// TwinCAT 3 PLC project Lamp
// Title: ESO LDC Lamp Library
// Company: ESO
// Author: Dan Popovic
// ProjectVersion: 1.1.1.6
// Description: Local Device Control - LDC Lamp Library based on State Machine
// ProgramVersion: 3.1.0.8
// libraries:
//   Tc2_Standard, * (Beckhoff Automation GmbH)
//   Tc2_System, * (Beckhoff Automation GmbH)
//   Tc3_EventLogger, * (Beckhoff Automation GmbH)
//   Tc3_Module, * (Beckhoff Automation GmbH)
//   VisuDialogs, * (System)
//   VisuSymbols,3.5.10.0,System
// project tree:
//   DUTs/Enumerated/ E_LAMP_COMMAND.TcDUT, E_LAMP_RPC_ERROR.TcDUT, E_LAMP_EVENT.TcDUT, E_LAMP_ERROR.TcDUT, E_LAMP_STATUS.TcDUT, E_LAMP_STATE.TcDUT, E_LAMP_HW_STATUS.TcDUT, E_LAMP_SUBSTATE.TcDUT
//   DUTs/Structures/ T_LAMP_CFG.TcDUT, T_SIM_LAMP_CFG.TcDUT, T_LAMP_CTRL.TcDUT, T_LAMP_INFO.TcDUT, T_LAMP_STAT.TcDUT, T_SIM_LAMP_STAT.TcDUT
//   / GlobalTextList.TcGTLO, PlcTask.TcTTO (not stored), Visualization Manager.TcVMO (not stored)
//   POUs/ FB_SIM_LAMP.TcPOU, FB_LAMP_BASE.TcPOU, FB_LAMP.TcPOU, MAIN.TcPOU
//   Version/ Global_Version.TcGVL
//   VISUs/ GUI_Lamp001.TcVIS, GUI_Lamp002.TcVIS
//   VISUs/Templates/ GUI_TEMPLATE_LAMP.TcVIS
// real-time tasks:
//   TASK PlcTask: cycle T#10ms, priority 20, ADS port 350
// variable links:
//   Lamp/Lamp Instance <-> Lamp/Lamp Instance
//     PlcTask Inputs/MAIN.Lamp001.i_bFault <-> PlcTask Outputs/MAIN.SIM_Lamp001.q_bFault
//     PlcTask Inputs/MAIN.Lamp002.i_bFault <-> PlcTask Outputs/MAIN.SIM_Lamp002.q_bFault
//     PlcTask Inputs/MAIN.Lamp001.i_bOn <-> PlcTask Outputs/MAIN.SIM_Lamp001.q_bOn
//     PlcTask Inputs/MAIN.Lamp002.i_bOn <-> PlcTask Outputs/MAIN.SIM_Lamp002.q_bOn
//     PlcTask Inputs/MAIN.Lamp001.i_nCouplerState <-> PlcTask Outputs/MAIN.SIM_Lamp001.q_nCouplerState
//     PlcTask Inputs/MAIN.Lamp002.i_nCouplerState <-> PlcTask Outputs/MAIN.SIM_Lamp002.q_nCouplerState
//     PlcTask Inputs/MAIN.Lamp001.i_nOn <-> PlcTask Outputs/MAIN.SIM_Lamp001.q_nOn
//     PlcTask Inputs/MAIN.Lamp002.i_nOn <-> PlcTask Outputs/MAIN.SIM_Lamp002.q_nOn
//     PlcTask Inputs/MAIN.SIM_Lamp001.i_bSwitch <-> PlcTask Outputs/MAIN.Lamp001.q_bSwitch
//     PlcTask Inputs/MAIN.SIM_Lamp002.i_bSwitch <-> PlcTask Outputs/MAIN.Lamp002.q_bSwitch

// ---- DUTs/Enumerated/E_LAMP_COMMAND.TcDUT
{attribute 'qualified_only'}
{attribute 'strict'}
TYPE E_LAMP_COMMAND :
(
	NONE	:= 0,
	
	RESET,
	INIT,
	STOP,
	ENABLE,
	DISABLE,
	ON,
	OFF
	
);
END_TYPE

// ---- DUTs/Enumerated/E_LAMP_RPC_ERROR.TcDUT
{attribute 'qualified_only'}
{attribute 'strict'}
TYPE E_LAMP_RPC_ERROR :
(
	OK						:= 0,
	NOT_OP					:= -1,			
	NOT_NOTOP_READY			:= -2,			
	NOT_NOTOP_NOTREADY		:= -3,			
	SWITCHING_ON			:= -4,			
	SWITCHING_OFF			:= -5,			
	COOLING					:= -6,			
	LOCAL					:= -7			
);
END_TYPE

// ---- DUTs/Enumerated/E_LAMP_EVENT.TcDUT
{attribute 'qualified_only'}
{attribute 'strict'}
TYPE E_LAMP_EVENT :
(
	NONE	:= 0,
	
	(* events corresponding to commands *)
	RESET,
	INIT,
	STOP,
	ENABLE,
	DISABLE,
	ON,
	OFF,
	
	(* 
		Events corresponding to internal events 
	*)
	
	INITON,		// Needed for detection of HW failures during initialisation
	INITOFF,
	DISABLEON,
	DISABLEOFF,
	WARMED_UP,
	COOLED_DOWN,
	LIMIT_ON,	// Time ON limit has been exceeded
	
	(* events mapped to HW signals *)
	ISON,
	ISOFF,

	HWOK,
	ERRHW,
	ERRMAXON,
	ERRFAULT,
	ERRINIT,
	ERRDISABLE,
	ERRTIMEOUTOFF,
	ERRTIMEOUTON
	
);
END_TYPE

// ---- DUTs/Enumerated/E_LAMP_ERROR.TcDUT
{attribute 'qualified_only'}
{attribute 'strict'}
TYPE E_LAMP_ERROR :
(
	OK					:= 0,
	HW_NOT_OP,			
	INIT_FAILURE,		
	UNEXPECTED_OFF,
	UNEXPECTED_ON,
	FAULT_SIG,
	MAXON,
	STILL_COOLING,
	TIMEOUT_DISABLE,
	TIMEOUT_INIT,
	TIMEOUT_OFF,
	TIMEOUT_ON,
	// Simulator errors
	SIM_NOT_INITIALISED	:= 90,
	SIM_NULL_POINTER		:= 100	
);
END_TYPE

// ---- DUTs/Enumerated/E_LAMP_STATUS.TcDUT
{attribute 'qualified_only'}
{attribute 'strict'}
TYPE E_LAMP_STATUS :
(
	OK	:= 0,
	ERROR
);
END_TYPE

// ---- DUTs/Enumerated/E_LAMP_STATE.TcDUT
{attribute 'qualified_only'}
{attribute 'strict'}
TYPE E_LAMP_STATE :
(
	NONE	:= 0,
	NOTOP,
	OP
);
END_TYPE

// ---- DUTs/Enumerated/E_LAMP_HW_STATUS.TcDUT
{attribute 'qualified_only'}
{attribute 'strict'}
TYPE E_LAMP_HW_STATUS :
(
	UNKNOWN	:= 0,
	ERROR,
	OFF,
	ON
);
END_TYPE

// ---- DUTs/Enumerated/E_LAMP_SUBSTATE.TcDUT
{attribute 'qualified_only'}
{attribute 'strict'}
TYPE E_LAMP_SUBSTATE :
(
	NONE				:= 0,
	
	NOTOP_NOTREADY		:= 100,
	NOTOP_INITIALIZING	:= 102,
	NOTOP_READY_OFF		:= 103,
	NOTOP_READY_ON		:= 104,
	NOTOP_ERROR			:= 199,
	
	OP_DISABLING		:= 205,
	OP_OFF				:= 206,            
	OP_SWITCHING_OFF	:= 207,           
	OP_COOLING			:= 208,
	OP_ON				:= 209,
	OP_SWITCHING_ON		:= 210,
	OP_WARMING			:= 211,
	OP_ERROR			:= 299
);
END_TYPE

// ---- DUTs/Structures/T_LAMP_CFG.TcDUT
TYPE T_LAMP_CFG :
STRUCT
	sName:				STRING	:= 'Lamp';	// Instance name
	bActiveLowFault:	BOOL 	:= FALSE;	(* If TRUE, Fault signal is Active Low *)
	bActiveLowOn:		BOOL 	:= FALSE;	(* If TRUE, On signal is Active Low *)
	bActiveLowSwitch:	BOOL 	:= FALSE;	(* If TRUE, Switch ctrl signal is Active Low *)

	bIgnoreFault:		BOOL 	:= FALSE;	(* If TRUE, Fault feedback signal is ignored *)
	bInitialState:		BOOL 	:= FALSE;	(* default lamp state is OFF *)
	bInvertAnalog:		BOOL 	:= FALSE;	(* If TRUE, analog feedback is active, if signal < nAnalogThreshold *)
	
	lrInitialIntensity:	LREAL 	:= 0.0;		// Initial intensity [%]. Default 0.0.

	nAnalogThreshold:	DINT 	:= 0;		(* Analog feedback signal threshold [bits].
										  	If this signal is used, any value above it will indicate that the lamp is ON. *)
	nFullRange:			UDINT 	:= 32767;	(* Full range of A/D converter for analog output for intensity control. Default is 15-bit.
										  	Beckhoff 16-bit analog output terminals include the sign.
										  	Effectively, for 0-10V terminals, this is a 15-bit resolution.  *)
	nSigStablePeriod:   UDINT 	:= 100;		(* signal is stable if it has been constant for so long [msec] *)
	nTimeout:     		UDINT 	:= 3000;	(* timeout for transitions [msec] *)


	nCooldown:			UDINT 	:= 0;		(* Cooldown time [sec] *)
	nMaxOn:				UDINT 	:= 0;		(* Maximum time for lamp to be ON [sec]. Zero means no limit. *)
	nWarmup:			UDINT 	:= 0;		(* Warmup time [sec] *)
	
	// Logging
	bLogExtTime:		BOOL 	:= FALSE;		// If TRUE, use external time in event logs. Default FALSE.
	bDebug:				BOOL 	:= FALSE;		// If TRUE, show event logs of Debug type. Default FALSE.
	bLog:				BOOL 	:= TRUE;		// If TRUE, log events. Default TRUE.
	
END_STRUCT
END_TYPE

// ---- DUTs/Structures/T_SIM_LAMP_CFG.TcDUT
TYPE T_SIM_LAMP_CFG :
STRUCT
	bActiveLowFault:	BOOL := FALSE;
	bActiveLowOn:		BOOL := FALSE;
	bActiveLowSwitch:	BOOL := FALSE;

	bInvertAnalog:		BOOL := FALSE;	// If TRUE, analog feedback is active, if signal < nAnalogThreshold
	
	nAnalogThreshold:	DINT := 0;		// Analog feedback signal threshold [bits].
	nDelay:     		UDINT := 1000;	// Simulated delay for commands [msec]
	
END_STRUCT
END_TYPE

// ---- DUTs/Structures/T_LAMP_CTRL.TcDUT
TYPE T_LAMP_CTRL :
STRUCT
	nCommand:		E_LAMP_COMMAND	:= E_LAMP_COMMAND.NONE;	(* See E_LAMP_COMMAND *)
	lrIntensity: 	LREAL	:= 0.0;					(* Intensity 0-100% [%] *)
	nTimeOnLimit:	UDINT	:= 0;					(* Auto OFF after this time [sec]. 0 - no limit *)
	bExecute:		BOOL;
	
END_STRUCT
END_TYPE

// ---- DUTs/Structures/T_LAMP_INFO.TcDUT
TYPE T_LAMP_INFO :
STRUCT
(*
Driver Information 

Change Log:
	0.1	2016-07-07	- First version.
	0.2	2016-07-08	- Implemented warming up and cooling down.
					- Creation of Lamp.library.
					- Cleanup of code.
	0.3	2016-07-11	- Implemented time ON/OFF update.
					- Implemented MAXON protection.
	0.4	2016-07-11	- Addition of Configuration and Status in Template GUI.
					- Addition of Local Control in Template GUI.
	0.5	2016-07-11	- GUI buttons disabled if not in Local Mode.
	0.6	2016-07-12	- Corrected Time Update.
					- Corrected error handling and display.
	0.7 2017-01-30	- Addition of stat.sLastCommand.
					- Adopted Simulator from VLT FB_SIM_LAMP.
	0.8 2017-09-04	- Removed METHOD ActionDisableComplete.
					- Re-odered config and status parameters.
					- Improved checks returned values in RPC calls.
					- Addition of input parameter in_lrIntensity to RPC_On().
	0.9.0.0			- Single pointer to simulator
					- Updated Visualisation version
	0.10.0.0		- Simulator pointer renamed to ptrDev.
					- Additional checks in RPC_On/Off.
	0.11.0.0		- Corrected handling of intensity.
					- Addition of RPC Call Status in GUI template.
	0.12.0.0		- Corrected Simulator handling of Update.
					- Removed bUpdate variable from Simulator.
					- Errors cleared on ON and OFF commands.
	0.13.0.0		- Addition of all cfg params as input params.
					- Addition of M_Configure() in FB_LAMP_BASE.
					- Added return value for Simulator RPC calls.
					- Added small delay to simulator on re-boot.
					- Moved sName to cfg structure.
	0.14.0.0		- Addition of stat.sLibVersion
	0.15.0.0		- RPC calls return INT.
					- Addition of E_LAMP_RPC_ERROR.
	0.16.0.0		- Addition of M_GetErrorText().
					- M_SetStatus() replaced SetStatus().
					- Improved error handling.
	0.17.0.0		- Addition of M_GetRpcErrorText().
					- Addition of M_SetRpcStatus().
					- Improved template GUI.
	0.18.0.0		- Improved the State Machine to reflect HW State.
	0.18.0.1		- Tc2_System.F_GetSystemTime() used in GetTimeInSec().
					- Addition of library category ESO/ELT.
	0.19.0.0		- Renaming States STANDBY->NOTOP & FAILURE->ERROR.
					- RPC commands rejected in Local mode.
	0.20.0.0		- Addition of nTimeOnLimit control parameter.
	1.0.0.0			- WARNING: Requires TwinCAT 3.1 build 4022.20 or higher.
					- Projects need Tc3_EventLogger library included in References.
					- Addition of Methods for Event Logs.
					- Addition of method RPC_Debug().
	1.0.0.1			- Addition of cfg.bLog flag for enable/disable of logging.
					- Renamed RPC_Debug() to RPC_SetDebug().
					- Addition of RPC_SetLog().
	1.0.0.2			- Addition of {attribute 'OPC.UA.DA':='0'} before in_bLog declaration.
	1.0.0.3			- Compiled with TwinCAT 3.1 build 4022.27.
					- Renamed TC_EVENTS.OpsEventClass to TC_EVENTS.LampOpsEventClass.
					- Solved problem of 'growing' libraries by setting Property/Advanced/BuildAction to None for Lamp.library.
	1.1.0.0			- Using Strict enumerations.
*)
	sDate:			STRING(32)	:= '2019-04-24';
	sDescription:	STRING(80) 	:= 'State Machine based Lamp controller';
	sName:			STRING(64)	:= 'FB_LAMP';
	sPlatform:		STRING(32)	:= 'CoDeSys';
	sSynopsis:		STRING(64)	:= 'State Machine based Lamp controller';
	nVersionMajor:	DINT		:= 1;
	nVersionMinor:	DINT		:= 1;
END_STRUCT
END_TYPE

// ---- DUTs/Structures/T_LAMP_STAT.TcDUT
TYPE T_LAMP_STAT :
STRUCT
	//
	// Common variables START
	//
	bLocal:			BOOL	:= FALSE;						(* if TRUE, device operated from PLC GUI *)
	bCheckTimeLeft:	BOOL	:= FALSE;						(* if TRUE, check for max time is active *)
	bOnAnalog:		BOOL	:= FALSE;						(* if TRUE, analog  ON is active *)
	bOnDigital:		BOOL	:= FALSE;						(* if TRUE, digital ON is active *)

	nOn:			DINT		:= 0;		// Analog feedback [bit]
	
	nLastCommand:	E_LAMP_COMMAND	:= E_LAMP_COMMAND.NONE;		(* Last command sent to the device *)

	nErrorCode: 	E_LAMP_ERROR 	:= E_LAMP_ERROR.HW_NOT_OP;	(* Error code *)
	nHwStatus: 		E_LAMP_HW_STATUS:= E_LAMP_HW_STATUS.UNKNOWN;(* Unknown, error, on, of. See E_LAMP_HW_STATUS *)
	nRpcErrorCode: 	E_LAMP_RPC_ERROR:= E_LAMP_RPC_ERROR.OK;		(* RPC Error code *)
	nStatus: 		E_LAMP_STATUS	:= E_LAMP_STATUS.ERROR; 	(* Device status *)

	sErrorText: 	STRING 	:= 'OK'; 						(* Error text *)
	sHwStatus: 		STRING 	:= 'UNKNOWN'; 					(* HW Status in textual form: 'UNKNOWN', 'ERROR', 'OPEN' or 'CLOSED' *)
	sLastCommand:	STRING	:= 'NONE';						(* Last command, as string, sent to the device *)
	sLibVersion:	STRING	:= 'UNKNOWN';					(* Library version as string, e.g. '1.2.0.0' *)
	sRpcErrorText: 	STRING 	:= 'OK'; 						(* RPC Error text *)
	sStatus: 		STRING 	:= 'OK'; 						(* Status in textual form, e.g. 'OFF' *)
	
	sState:			STRING	:= 'NOT OP';
	sSubstate:		STRING	:= 'NOT READY';
	
	nState:			E_LAMP_STATE	:= E_LAMP_STATE.NOTOP;
	nSubstate:		E_LAMP_SUBSTATE	:= E_LAMP_SUBSTATE.NOTOP_NOTREADY;
	
	sActionDesc:	STRING	:= '';
	sEventDesc:		STRING	:= '';

	nCycleCounter:	UDINT	:= 0;							// Alive flag
	nCycleTime:		UDINT	:= 0;							// Cycle time in us (microsec)
	//
	// Common variables END
	//
	
	//
	// Device specific variables
	//
	lrIntensity: 		LREAL	:= 0.0; 	(* Intensity: 0-100% [%]*)

	nTimeLeft: 			UDINT 	:= 777;		(* Remaining Time before lamp is switched OFF [sec]. 777 means no limit. *)
	nTimeOn: 			UDINT 	:= 0;		(* Time lamp has been ON since last ON command [sec] *)
	nTimeOnLimit:		UDINT	:= 0;		(* Auto OFF after this time [sec]. 0 - no limit *)
	nTimeOnStart:		UDINT 	:= 0;		(* Absolute start time of last lamp ON command [sec] *)
	nTimeOnTotal:		UDINT 	:= 0;		(* Total time lamp has been ON [sec] *)
	nTimeOnTotalStart:	UDINT 	:= 0;		(* Absolute start time of lamp ON [sec] *)
	nTimeOff: 			UDINT 	:= 0;		(* Time lamp has been OFF [sec] *)
	nTimeOffStart:		UDINT 	:= 0;		(* Time lamp has been OFF [sec] *)
END_STRUCT
END_TYPE

// ---- DUTs/Structures/T_SIM_LAMP_STAT.TcDUT
TYPE T_SIM_LAMP_STAT :
STRUCT
	bInitialised:	BOOL	:= FALSE;						(* If TRUE, lamp simulator is initialised *)

	nErrorCode: 	E_LAMP_ERROR 	:= E_LAMP_ERROR.SIM_NOT_INITIALISED;	(* Error code *)
	sErrorText: 	STRING 	:= 'NOT INITIALISED'; 			(* Error text *)
	sStatus: 		STRING 	:= 'ERROR'; 					(* Lamp status in textual form, e.g. 'OFF' *)
END_STRUCT
END_TYPE

// ---- Version/Global_Version.TcGVL
{attribute 'TcGenerated'}
{attribute 'no-analysis'}
{attribute 'linkalways'}
// This function has been automatically generated from the project information.
VAR_GLOBAL CONSTANT
	{attribute 'const_non_replaced'}
	stLibVersion_ESO_LDC_Lamp_Library : ST_LibVersion := (iMajor := 1, iMinor := 1, iBuild := 1, iRevision := 6, nFlags := 0, sVersion := '1.1.1.6');
END_VAR

// ---- POUs/FB_SIM_LAMP.TcPOU
FUNCTION_BLOCK FB_SIM_LAMP
VAR_INPUT
	ptrDev:		POINTER TO FB_LAMP;
END_VAR
VAR_OUTPUT
END_VAR
VAR
	ptrCfg:		POINTER TO T_LAMP_CFG;
	ptrStat:	POINTER TO T_LAMP_STAT;

	{attribute 'OPC.UA.DA':='1'}
	cfg:			T_SIM_LAMP_CFG;		(* ActiveLow configuration for each signal *)
	{attribute 'OPC.UA.DA':='1'}
	stat:			T_SIM_LAMP_STAT;	(* Simulator status parameters *)
	
	{attribute 'OPC.UA.DA':='0'}
	bSwitch:		BOOL := FALSE;
	{attribute 'OPC.UA.DA':='0'}
	bSwitchLast:	BOOL := FALSE;
	
	{attribute 'OPC.UA.DA':='0'}
	bOn:			BOOL := TRUE;	// Digital feedback
	{attribute 'OPC.UA.DA':='0'}
	nOn:			DINT := 0;		// Analog feedback
	{attribute 'OPC.UA.DA':='0'}
	bFault:			BOOL := FALSE;
	{attribute 'OPC.UA.DA':='0'}
	nCouplerState:	UINT := 8;       // normal coupler state
	
    (* Inputs *)
	{attribute 'OPC.UA.DA':='0'}
	i_bSwitch 		AT %I*: 	BOOL;

	(* Outputs *)	
	{attribute 'OPC.UA.DA':='0'}
	q_bFault 		AT %Q*: 	BOOL;
	{attribute 'OPC.UA.DA':='0'}
	q_bOn 			AT %Q*: 	BOOL;	// Digital feedback signal
	{attribute 'OPC.UA.DA':='0'}
	q_nOn 			AT %Q*: 	INT;	// Analog feedback signal
	{attribute 'OPC.UA.DA':='0'}
	q_nCouplerState AT %Q*:		UINT := 8;
	
	{attribute 'OPC.UA.DA':='0'}
	timer:			TON;
	
	{attribute 'OPC.UA.DA':='0'}
	trigger:		R_TRIG;	// To capture device INIT

	{attribute 'OPC.UA.DA':='0'}
	counter:		DINT	:= 0; 	// Counter used to 	

	{attribute 'OPC.UA.DA':='0'}
	nOnStart:		DINT;
	{attribute 'OPC.UA.DA':='0'}
	nOnEnd:			DINT;
	{attribute 'OPC.UA.DA':='0'}
	nOnDelta:		DINT;		// Total analog signal change during ramp
	
	t1, t2:	LREAL;

END_VAR

// Give simulator 20 cycles of idle until real device is ready.
IF counter < 20 THEN
	counter	:= counter + 1;
	RETURN;
END_IF

// Initialise the simulator, i.e. set pointers to the real device, etc.
IF NOT stat.bInitialised THEN
	ptrCfg	:= ADR(ptrDev^.cfg);
	ptrStat	:= ADR(ptrDev^.stat);

	// Check for NULL pointers in input parameters
	IF ptrCfg = 0  OR  ptrStat = 0 THEN
		stat.nErrorCode	:= E_LAMP_ERROR.SIM_NULL_POINTER;
		stat.sErrorText	:= 'ERROR: Input parameter is a NULL pointer';
		stat.sStatus	:= 'ERROR';
		RETURN;
	END_IF

	RPC_ResetConfig();	// Copy configuration from device
	
	// Set analog feedback to a good starting level.
	M_SetAnalogFeedback();

	timer(IN:=FALSE);
	timer(IN:=TRUE,PT:=UDINT_TO_TIME(100));	// Update almost immediately

	stat.nErrorCode	:= E_LAMP_ERROR.OK;
	stat.sErrorText	:= 'OK';
	stat.sStatus	:= 'OK';
	
	stat.bInitialised	:= TRUE;
	RETURN;
END_IF

// There are two possible triggers: 
// 	- Detect device INIT (action = 'ActionInitExecute')
// 	- Activation of switch (change of i_bSwitch state)

// Check for INIT trigger
trigger(CLK:=(ptrStat^.sActionDesc = 'ActionInitExecute'));

// Get the state of control command
bSwitch := M_GetLogicalState(i_bSwitch, cfg.bActiveLowSwitch);

IF trigger.Q THEN
	timer(IN:=FALSE);
	RPC_ResetConfig();	// Copy configuration from device
	// Set analog feedback to a good starting level.
	M_SetAnalogFeedback();
ELSIF bSwitch <> bSwitchLast THEN
	ReloadConfig();	// Reload configuration from device
	
	// Switch value has changed. 
	bSwitchLast	:= bSwitch;

	// Delayed response
	timer(IN:=FALSE);
	timer(IN:=TRUE,PT:=UDINT_TO_TIME(cfg.nDelay));
	
	// If analog feedback is used, find out how much to ramp it.
	IF cfg.nAnalogThreshold <> 0	THEN
		nOnStart	:= nOn;
		// Set target feedback is 10 bit beyond the threshold.
		// This value depends on the command (on/off) and the logic (over/under threshold).
		IF bSwitch = M_GetLogicalState(TRUE, cfg.bActiveLowSwitch) THEN
		// The command was ON
			IF cfg.bInvertAnalog THEN
				nOnEnd	:= cfg.nAnalogThreshold - 10;
			ELSE
				nOnEnd	:= cfg.nAnalogThreshold + 10;
			END_IF
		ELSE
		// The command was OFF
			IF cfg.bInvertAnalog THEN
				nOnEnd	:= MAX(32000, cfg.nAnalogThreshold + 10);	// was cfg.nAnalogThreshold + 10;
			ELSE
				nOnEnd	:= 0;	// was cfg.nAnalogThreshold - 10;
			END_IF
		END_IF
		// This is how much to change simulated feedback over cfg.nDelay.
		nOnDelta	:= nOnEnd - nOnStart;
	END_IF
END_IF


// Execute the timer
timer();

// If analog feedback is used, ramp up/down the simulated feedback.
IF cfg.nAnalogThreshold <> 0	THEN
	bOn	:= FALSE;	// Don't use the digital feedback.
	IF timer.ET > INT_TO_TIME(0)	THEN
		t1	:= TIME_TO_LREAL(timer.ET);
		t2	:= TIME_TO_LREAL(timer.PT);
		nOn	:=	nOnStart + LREAL_TO_INT((t1*t1*t1) / (t2*t2*t2) * nOnDelta);
	END_IF
ELSE
	nOn	:= 0;
END_IF

// Set new outputs once the timer has expired
IF timer.Q THEN
	timer(IN:=FALSE);	// Reset timer
	// Set digital output, i.e. feedback, if analog feedback is not used.
	IF cfg.nAnalogThreshold = 0	THEN
		bOn	:= M_GetLogicalState(bSwitch,	cfg.bActiveLowOn);
	END_IF
END_IF


(* Assign outputs *)
q_bFault		:= M_GetLogicalState(bFault, cfg.bActiveLowFault);
q_bOn 			:= bOn;
q_nOn			:= DINT_TO_INT(nOn);
q_nCouplerState := nCouplerState;

METHOD M_GetLogicalState : BOOL
(*
	This method returns the state of the variable based on its 
	activeLow configuration.
	Syntax:
		bState	:= M_GetLogicalState (<var value>,  <activeLow cfg>);
		
	Example 1:
		var = TRUE;
		activeLow = FALSE;
		bState	:= M_GetLogicalState (TRUE,  FALSE); = TRUE

	Example 2:
		var = TRUE;
		activeLow = TRUE;
		bState	:= M_GetLogicalState (TRUE,  TRUE); = FALSE
*)
VAR_INPUT
	state:		BOOL;
	activeLow:	BOOL;
END_VAR
IF activeLow THEN
	M_GetLogicalState := NOT state;
ELSE
	M_GetLogicalState := state;
END_IF
END_METHOD

// Set starting analog feedback depending 
// on the analog feedback configuration and the command.
METHOD M_SetAnalogFeedback
VAR_INPUT
END_VAR
// Reset analog feedback, if not used.
IF cfg.nAnalogThreshold = 0	THEN
	nOn	:= 0;
ELSE
	// Analog feedback set to a value equivalent to OFF.
	IF cfg.bInvertAnalog THEN
		nOn	:= MAX(32000, cfg.nAnalogThreshold + 10);
	ELSE
		nOn	:= 0;
	END_IF
END_IF
END_METHOD

METHOD ReloadConfig : BOOL
VAR_INPUT
END_VAR
cfg.bActiveLowOn		:= ptrCfg^.bActiveLowOn;
cfg.bActiveLowFault		:= ptrCfg^.bActiveLowFault;
cfg.bActiveLowSwitch	:= ptrCfg^.bActiveLowSwitch;
cfg.bInvertAnalog		:= ptrCfg^.bInvertAnalog;
cfg.nDelay				:= ptrCfg^.nTimeout / 2;	// Response delay = 1/2 of real lamp timeout
cfg.nAnalogThreshold	:= ptrCfg^.nAnalogThreshold;
nCouplerState			:= 8;

// Reset analog feedback, if not used.
IF cfg.nAnalogThreshold = 0	THEN
	nOn	:= 0;
END_IF
END_METHOD

{attribute 'TcRpcEnable':='1'}
METHOD RPC_ResetConfig : INT
VAR_INPUT
END_VAR
ReloadConfig();

// Set valid intensity feedback
nOn	:= cfg.nAnalogThreshold;


// Reset Fault signal
bFault		:= FALSE;

// Get the Switch value
bSwitch := M_GetLogicalState(i_bSwitch, cfg.bActiveLowSwitch);

bOn	:= M_GetLogicalState(bSwitch,	cfg.bActiveLowOn);	// Set lamp state

RPC_ResetConfig	:= E_LAMP_RPC_ERROR.OK;
END_METHOD

{attribute 'TcRpcEnable':='1'}
METHOD RPC_SetActiveLow_Fault : INT
VAR_INPUT
	bValue:	BOOL;
END_VAR
cfg.bActiveLowFault	:= bValue;

RPC_SetActiveLow_Fault	:= E_LAMP_RPC_ERROR.OK;
END_METHOD

{attribute 'TcRpcEnable':='1'}
METHOD RPC_SetActiveLow_On : INT
VAR_INPUT
	bValue:	BOOL;
END_VAR
cfg.bActiveLowOn	:= bValue;

RPC_SetActiveLow_On	:= E_LAMP_RPC_ERROR.OK;
END_METHOD

{attribute 'TcRpcEnable':='1'}
METHOD RPC_SetActiveLow_Switch : INT
VAR_INPUT
	bValue:	BOOL;
END_VAR
cfg.bActiveLowSwitch	:= bValue;

RPC_SetActiveLow_Switch	:= E_LAMP_RPC_ERROR.OK;
END_METHOD

{attribute 'TcRpcEnable':='1'}
METHOD RPC_SetCouplerState : INT
VAR_INPUT
	nValue:	UINT;
END_VAR
nCouplerState	:= nValue;

RPC_SetCouplerState	:= E_LAMP_RPC_ERROR.OK;
END_METHOD

{attribute 'TcRpcEnable':='1'}
METHOD RPC_SetDelay : INT
VAR_INPUT
	nDelay:	UDINT;
END_VAR
cfg.nDelay	:= nDelay;

RPC_SetDelay	:= E_LAMP_RPC_ERROR.OK;
END_METHOD

{attribute 'TcRpcEnable':='1'}
METHOD RPC_SetFault : INT
VAR_INPUT
	bValue:	BOOL;
END_VAR
bFault	:= bValue;

RPC_SetFault	:= E_LAMP_RPC_ERROR.OK;
END_METHOD

END_FUNCTION_BLOCK

// ---- POUs/FB_LAMP.TcPOU
FUNCTION_BLOCK FB_LAMP EXTENDS FB_LAMP_BASE
VAR_INPUT
END_VAR
VAR_OUTPUT
END_VAR
VAR
	
	(***** Local variables *****)
	{attribute 'OPC.UA.DA' := '0'}
	bOn:		BOOL;	(* Feedback - combination of digital and analog *)
	{attribute 'OPC.UA.DA' := '0'}
	bFault: 	BOOL;
	{attribute 'OPC.UA.DA' := '0'}
	toutCmd:	TON;
	{attribute 'OPC.UA.DA' := '0'}
	trg:		R_TRIG;
	{attribute 'OPC.UA.DA' := '0'}
	timer:		TON;	(* Timer for measuring duration of events *)
	


	(***** Physical signals - to be mapped!!! *****)

	(* Outputs *)
	{attribute 'OPC.UA.DA' := '0'}
	q_bSwitch 		AT %Q*: 		BOOL;	(* Lamp control digital output *)
	{attribute 'OPC.UA.DA' := '0'}
	q_nIntensity 	AT %Q*: 		INT;	(* Analog OUT [bit] *)

	(* Inputs *)	
	{attribute 'OPC.UA.DA' := '0'}
	i_nCouplerState	AT %I*: 		UINT;	(* Link it to Coupler->InfoData->State *)
	{attribute 'OPC.UA.DA' := '0'}
	i_bFault 		AT %I*: 		BOOL;	(* HW fault signal *)
	{attribute 'OPC.UA.DA' := '0'}
	i_bOn 			AT %I*: 		BOOL;	(* Digital feedback signal *)
	{attribute 'OPC.UA.DA' := '0'}
	i_nOn			AT %I*: 		INT;	(* Analog feedback signal *)

END_VAR

// Execute the base class object FB_LAMP_BASE
SUPER^();

METHOD ActionDisableExecute
VAR_INPUT
END_VAR
SetAction('ActionDisableExecute');

// Log event
M_LogEventStart('DISABLE');

(* Set Lamp initial state obtained from the configuration *)
q_bSwitch			:= M_GetLogicalState(cfg.bInitialState, cfg.bActiveLowSwitch);
stat.lrIntensity	:= cfg.lrInitialIntensity;
q_nIntensity		:= LREAL_TO_INT(stat.lrIntensity / 100.0 * cfg.nFullRange);

(* start the cmd timer *)
toutCmd(IN:=FALSE);
toutCmd(IN:=TRUE,PT:=UDINT_TO_TIME(cfg.nTimeout));
END_METHOD

METHOD ActionEnableComplete
VAR_INPUT
END_VAR
SetAction('ActionEnableComplete');

// Log event
M_LogEventEnd('ENABLE');

(* reply OK *)
M_SetStatus(E_LAMP_ERROR.OK);

(* Reset the timer action *)
toutCmd(IN:=FALSE);
END_METHOD

METHOD ActionErrExecute
VAR
END_VAR
SetAction('ActionErrExecute');

IF nEvent = E_LAMP_EVENT.ERRFAULT THEN
	M_SetStatus(E_LAMP_ERROR.FAULT_SIG);
END_IF
END_METHOD

METHOD ActionInitAbort
VAR_INPUT
END_VAR
SetAction('ActionInitAbort');

M_SetStatus(E_LAMP_ERROR.OK);

(* Reset the timer for the command *)
toutCmd(IN:=FALSE);
END_METHOD

METHOD ActionInitComplete
VAR_INPUT
END_VAR
SetAction('ActionInitComplete');

// Log event
M_LogEventEnd('INIT');

(* reply OK *)
M_SetStatus(E_LAMP_ERROR.OK);

(* Reset the timer action *)
toutCmd(IN:=FALSE);
END_METHOD

METHOD ActionInitExecute
VAR_INPUT
END_VAR
VAR
	nCurrentTime:	UDINT;
END_VAR
SetAction('ActionInitExecute');

// Log event
M_LogEventStart('INIT');

M_SetStatus(E_LAMP_ERROR.OK);	// Clear any error

nCurrentTime			:= M_GetTimeInSec();
stat.nTimeOffStart		:= nCurrentTime;
M_UpdateTimes(bOnState:=FALSE, bRestart:=FALSE, bReset:=FALSE);


(* Set Lamp initial state obtained from the configuration *)
q_bSwitch			:= M_GetLogicalState(cfg.bInitialState, cfg.bActiveLowSwitch);
IF NOT cfg.bInitialState	THEN
	cfg.lrInitialIntensity	:= 0.0;
END_IF
stat.lrIntensity	:= cfg.lrInitialIntensity;
q_nIntensity		:= LREAL_TO_INT(stat.lrIntensity / 100.0 * cfg.nFullRange);

(* start the cmd timer *)
toutCmd(IN:=FALSE);
toutCmd(IN:=TRUE,PT:=UDINT_TO_TIME(cfg.nTimeout));
END_METHOD

METHOD ActionInitReject
VAR_INPUT
END_VAR
SetAction('ActionInitReject');

(* Reject an INIT command since another one is in progress. *)
(* do not reset the timer ... *)
END_METHOD

METHOD ActionMaxOnFailure
VAR_INPUT
END_VAR
(* code to initiate the switching OFF of the lamp *)
SetAction('ActionMaxOnFailure');

// Log event
M_LogEventError('Max ON time exceeded. Lamp switched OFF.');

(* Set the error *)
M_SetStatus(E_LAMP_ERROR.MAXON);

M_UpdateTimes(bOnState:=FALSE, bRestart:=TRUE, bReset:=FALSE);


(* Switch lamp OFF *)
q_bSwitch			:= M_GetLogicalState(FALSE, cfg.bActiveLowSwitch);
stat.lrIntensity	:= 0;
q_nIntensity		:= 0;


(* 
	Reset signal trigger and its timer. 
	Next transition activity, e.g. ActivitySwitchingOff, will complete when the signal has been OFF 
	for longer than cfg.nSigStablePeriod [ms].
*)
trg(CLK:=FALSE);
timer(IN:=FALSE);	// Timer for stable signal lasting cfg.nSigStablePeriod

(* Restart the command timer *)
toutCmd(IN:=FALSE);
toutCmd(IN:=TRUE,PT:=UDINT_TO_TIME(cfg.nTimeout));
END_METHOD

METHOD ActionOffExecute
VAR_INPUT
END_VAR
(* code to initiate the switching OFF of the lamp *)
SetAction('ActionOffExecute');

// Log event
M_LogEventStart('OFF');

(* Clear the error *)
M_SetStatus(E_LAMP_ERROR.OK);

M_UpdateTimes(bOnState:=FALSE, bRestart:=TRUE, bReset:=FALSE);


(* Switch lamp OFF *)
q_bSwitch			:= M_GetLogicalState(FALSE, cfg.bActiveLowSwitch);
stat.lrIntensity	:= 0;
q_nIntensity		:= 0;

(* 
	Reset signal trigger and its timer. 
	Next transition activity, e.g. ActivitySwitchingOff, will complete when the signal has been OFF 
	for longer than cfg.nSigStablePeriod [ms].
*)
trg(CLK:=FALSE);
timer(IN:=FALSE);	// Timer for stable signal lasting cfg.nSigStablePeriod

(* Restart the command timer *)
toutCmd(IN:=FALSE);
toutCmd(IN:=TRUE,PT:=UDINT_TO_TIME(cfg.nTimeout));
END_METHOD

METHOD ActionOnExecute
VAR_INPUT
END_VAR
(* Code to initiate turning the lamp ON *)

SetAction('ActionOnExecute');

// Log event
M_LogEventStart('ON');

(* Clear the error *)
M_SetStatus(E_LAMP_ERROR.OK);

(* Turn the control signal ON  and set the intensity *)
q_bSwitch			:= M_GetLogicalState(TRUE, cfg.bActiveLowSwitch);
stat.lrIntensity	:= ctrl.lrIntensity;
q_nIntensity		:= LREAL_TO_INT(stat.lrIntensity / 100.0 * cfg.nFullRange);

// Save time limit for ON and clear it from the command parameters
stat.nTimeOnLimit	:= ctrl.nTimeOnLimit;
ctrl.nTimeOnLimit	:= 0;


(* 
	Reset signal trigger and its timer. 
	Next transition activity, e.g. ActivitySwitchingOn, will complete when the signal has been ON 
	for longer than cfg.nSigStablePeriod [ms].
*)
trg(CLK:=FALSE);
timer(IN:=FALSE);	// Timer for stable signal lasting cfg.nSigStablePeriod

(* Start the timer for command timeout of cfg.nTimeout *)
toutCmd(IN:=FALSE);	
toutCmd(IN:=TRUE,PT:=UDINT_TO_TIME(cfg.nTimeout));
END_METHOD

METHOD ActionResetExecute
VAR_INPUT
END_VAR
SetAction('ActionResetExecute');

// Log event
M_LogEventEnd('RESET');

(* reply Error *)
M_SetStatus(E_LAMP_ERROR.OK);

(* Disable outputs *)
q_bSwitch			:= FALSE;
stat.lrIntensity	:= 0;
q_nIntensity		:= 0;

// Reset ON/OFF times
M_UpdateTimes(bOnState:=bOn,bRestart:=FALSE,bReset:=TRUE);	

(* Reset the timer for the command *)
toutCmd(IN:=FALSE);
END_METHOD

METHOD ActionUnexpExecute
VAR
END_VAR
SetAction('ActionUnexpExecute');

IF nEvent = E_LAMP_EVENT.ISON THEN
	// In case of a timeout while switching to ON the state after the timeout
	// will be E_LAMP_SUBSTATE.OP_OFF and later on the lamp will go ON. 
	// In this case, we don't want to set
	// the error to E_LAMP_ERROR.UNEXPECTED_ON but rather scilently
	// change the state to E_LAMP_SUBSTATE.OP_ON.
	IF 	stat.nErrorCode <> E_LAMP_ERROR.TIMEOUT_ON  AND
		stat.nErrorCode <> E_LAMP_ERROR.TIMEOUT_OFF 	THEN
		M_LogEventGeneral('Lamp unexpectedly switched ON');
		M_SetStatus(E_LAMP_ERROR.UNEXPECTED_ON);
	END_IF
ELSIF nEvent = E_LAMP_EVENT.ISOFF THEN
	// In case of a timeout while switching to OFF the state after the timeout
	// will be E_LAMP_SUBSTATE.OP_ON and later on the lamp will go OFF. 
	// In this case, we don't want to set
	// the error to E_LAMP_ERROR.UNEXPECTED_OFF but rather scilently
	// change the state to E_LAMP_SUBSTATE.OP_OFF.
	IF 	stat.nErrorCode <> E_LAMP_ERROR.TIMEOUT_OFF	AND
		stat.nErrorCode <> E_LAMP_ERROR.TIMEOUT_ON THEN
		M_LogEventGeneral('Lamp unexpectedly switched OFF');
		M_SetStatus(E_LAMP_ERROR.UNEXPECTED_OFF);
	END_IF
ELSIF nEvent = E_LAMP_EVENT.ON THEN
	// Clear time limit from the command parameters
	ctrl.nTimeOnLimit	:= 0;
	M_SetStatus(E_LAMP_ERROR.STILL_COOLING);
END_IF
END_METHOD

METHOD ActivityCoolingDown
VAR_INPUT
END_VAR
(* 
	This activity waits for cfg.nCooldown seconds until the lamp has warmed up.
	It triggers E_LAMP_EVENT.WARMED_UP event. 
*)
SetAction('ActivityCoolingDown');

// Update the OFF time
M_UpdateTimes(bOnState:=FALSE, bRestart:=FALSE, bReset:=FALSE);

(* 
	Warming is complete on expiration of the timer.
	If there is no warmup (cfg.nWarmup = 0), just set the event E_LAMP_EVENT.WARMED_UP.
*)
toutCmd();
IF 	toutCmd.Q OR 
	cfg.nCooldown = 0 OR
	(cfg.nCooldown > 0 AND stat.nTimeOff > cfg.nCooldown)	THEN
	// Log event
	M_LogEventEnd('OFF');

	toutCmd(IN:=FALSE);	(* Reset Timer *)
	
	nInternalEvent 		:= E_LAMP_EVENT.COOLED_DOWN;	// This will bring us to (E_LAMP_STATE.OP, E_LAMP_SUBSTATE.OP_OFF)
END_IF
END_METHOD

METHOD ActivityDisabling
VAR_INPUT
END_VAR
(* 
	Activity to monitor the lamp disabling task. 
	The end state should be the predefined position of the lamp
	that is defined by configuration parameter cfg.bInitialState.
*)
SetAction('ActivityDisabling');

(* check if the initial position is reached *)
IF cfg.bInitialState = FALSE THEN
	(* Waiting for OFF state *)
	IF	bOn   = FALSE THEN
		// Log event
		M_LogEventEnd('DISABLE_OFF');

		nEvent  := E_LAMP_EVENT.DISABLEOFF;
		M_SetStatus(E_LAMP_ERROR.OK);
		RETURN;
	END_IF
ELSE
	(* Waiting for ON state *)
	IF	bOn   = TRUE  THEN
		// Log event
		M_LogEventEnd('DISABLE_ON');

		nEvent  := E_LAMP_EVENT.DISABLEON;
		M_SetStatus(E_LAMP_ERROR.OK);
		RETURN;
	END_IF		
END_IF


(* 
	if the timeout is detected before reaching the target position, 
	then trigger the internal error event 
*)
toutCmd(IN:=TRUE);
IF toutCmd.Q THEN
	// Log event
	M_LogEventError('DISABLE command timed out');

	toutCmd(IN:=FALSE);	(* Reset the timer *)
	nInternalEvent  := E_LAMP_EVENT.ERRDISABLE;
	SetEvent(E_LAMP_ERROR.TIMEOUT_DISABLE);
END_IF
END_METHOD

METHOD ActivityInitializing
VAR_INPUT
END_VAR
(* 
	Activity to monitor the Lamp initialization task and 
	trigger the E_LAMP_EVENT.INITOFF or E_LAMP_EVENT.INITON event depending 
	on the configured default state. 		
*)
SetAction('ActivityInitializing');


(* 
	Check if the initial position is reached.
	We need additional internal events E_LAMP_EVENT.INITOFF & E_LAMP_EVENT.INITON in order to
	cope with the scenario when the initial state is the oposit one from the configured target.
	Example:
		The Lamp ISOFF at the beginning of this activity while the configured default state ISOFF.
		By introducing E_LAMP_EVENT.INITOFF & E_LAMP_EVENT.INITON we avoid the ISOFF event.
*)
IF cfg.bInitialState = FALSE THEN
	(* Waiting for OFF state *)
	IF	bOn   = FALSE THEN
		nInternalEvent  := E_LAMP_EVENT.INITOFF;
	END_IF
ELSE
	(* Waiting for ON state *)
	IF	bOn   = TRUE  THEN
		nInternalEvent  := E_LAMP_EVENT.INITON;
	END_IF		
END_IF


(* 
	If the timeout is detected before reaching the initial position, 
	then trigger the internal error event 
*)
toutCmd(IN:=TRUE);
IF toutCmd.Q THEN
	// Log event
	M_LogEventError('INIT command timed out');

	toutCmd(IN:=FALSE);	(* Reset the timer *)
	nInternalEvent  := E_LAMP_EVENT.ERRINIT;
	SetEvent(E_LAMP_ERROR.TIMEOUT_INIT);
END_IF
END_METHOD

METHOD ActivityOff
VAR_INPUT
END_VAR
SetAction('ActivityOff');

// Clear time limit for ON from the status
stat.nTimeOnLimit	:= 0;

// Update the OFF time
M_UpdateTimes(bOnState:=FALSE, bRestart:=FALSE, bReset:=FALSE);
END_METHOD

METHOD ActivityOn
VAR_INPUT
END_VAR
SetAction('ActivityOn');

// Update the ON time
M_UpdateTimes(bOnState:=TRUE, bRestart:=FALSE, bReset:=FALSE);

// Check if the lamp has been ON longer than the time limit for that command.
IF stat.nTimeOnLimit > 0 AND stat.nTimeOn > stat.nTimeOnLimit THEN
	M_LogEventGeneral('Time ON limit reached. Switching lamp OFF.');
	nEvent  := E_LAMP_EVENT.LIMIT_ON;
	RETURN;
END_IF
END_METHOD

METHOD ActivitySwitchingOff
VAR_INPUT
END_VAR
(* 
	This activity monitors the OFF lamp task and 
	triggers the ISOFF event at completion. 
*)
SetAction('ActivitySwitchingOff');


(* 
	The signal has to be OFF for longer than cfg.nSigStablePeriod [msec].
	The timer will start when bOn=FALSE trigger is detected.
*)
(* Execute trigger - note the 'NOT bOn' detectiong the transition from ON to OFF *)
trg(CLK := NOT bOn);

IF trg.Q THEN
	(* Restart the signal duration timer *)
	timer(IN:=FALSE);
	timer(IN:=TRUE,PT:=UDINT_TO_TIME(cfg.nSigStablePeriod));
END_IF

(* Execute signal duration timer *)
timer();

IF	timer.Q OR 
	((NOT bOn) AND cfg.nSigStablePeriod = 0) THEN
	timer(IN:=FALSE);	// Reset the signal duration timer
	toutCmd(IN:=FALSE);	// Reset the command timeout timer

	(* Update time ON/OFF *)
	M_UpdateTimes(bOnState:=TRUE, bRestart:=FALSE, bReset:=FALSE);

	(* 
		Normally, we would go to state E_LAMP_SUBSTATE.OP_COOLING. 
		However, if the cooldown time is zero, i.e. no cooldown, we go directly to state E_LAMP_SUBSTATE.OP_OFF.
	*)
	IF cfg.nCooldown > 0 THEN
		// Log event
		M_LogEventStart('COOLING');

		// Restart the command timeout timer
		toutCmd(IN:=TRUE,PT:=UDINT_TO_TIME(cfg.nCooldown * 1000));	// [sec] => [msec]
		nInternalEvent 		:= E_LAMP_EVENT.ISOFF;	// This will bring us to SetState(E_LAMP_STATE.OP, E_LAMP_SUBSTATE.OP_COOLING)
	ELSE
		// Log event
		M_LogEventEnd('OFF');

		nInternalEvent 		:= E_LAMP_EVENT.COOLED_DOWN;	// This will bring us to SetState(E_LAMP_STATE.OP, E_LAMP_SUBSTATE.OP_OFF)
	END_IF
	
//	M_SetStatus(E_LAMP_ERROR.OK);	

	RETURN;
END_IF

(* 
	if the timeout is detected before reaching the position, 
	then trigger the internal error event 
*)
toutCmd();
IF toutCmd.Q THEN
	toutCmd(IN:=FALSE);	(* Reset Timer *)
	timer(IN:=FALSE);	(* Reset the signal duration timer *)
	
	nInternalEvent  := E_LAMP_EVENT.ERRTIMEOUTOFF;
	SetEvent(E_LAMP_EVENT.ERRTIMEOUTOFF);
	M_SetStatus(E_LAMP_ERROR.TIMEOUT_OFF);	
END_IF
END_METHOD

METHOD ActivitySwitchingOn
VAR_INPUT
END_VAR
(* 
	This activity to monitor the ON lamp task and 
	trigger the ISON event at completion. 
*)
SetAction('ActivitySwitchingOn');

(* 
	The signal has to be ON for longer than cfg.nSigStablePeriod [msec].
	The timer will start when bOn trigger is detected.
*)
(* Execute trigger *)
trg(CLK:=bOn);

IF trg.Q THEN
	(* Restart the signal duration timer *)
	timer(IN:=FALSE);
	timer(IN:=TRUE,PT:=UDINT_TO_TIME(cfg.nSigStablePeriod));
END_IF

(* Execute signal duration timer *)
timer();

IF	timer.Q OR 
	(bOn AND cfg.nSigStablePeriod = 0) THEN
	timer(IN:=FALSE);	// Reset the signal duration timer
	toutCmd(IN:=FALSE);	// Reset the command timeout timer

	(* Update time ON/OFF *)
	IF stat.nTimeOn > 0 THEN
		// Lamp was already ON, restart the ON time.
		M_UpdateTimes(bOnState:=TRUE, bRestart:=TRUE, bReset:=FALSE);
	ELSE
		// Lamp was OFF, don't restart the ON time.
		M_UpdateTimes(bOnState:=TRUE, bRestart:=FALSE, bReset:=FALSE);
	END_IF

	(* 
		Normally, we would go to state E_LAMP_SUBSTATE.OP_WARMING. 
		However, if the warmup time is zero, i.e. no warmup, we go directly to state E_LAMP_SUBSTATE.OP_ON.
	*)
	IF cfg.nWarmup > 0 THEN
		// Log event
		M_LogEventStart('WARMING UP');

		// Restart the command timeout timer
		toutCmd(IN:=TRUE,PT:=UDINT_TO_TIME(cfg.nWarmup * 1000));	// [sec] => [msec]
		nInternalEvent 		:= E_LAMP_EVENT.ISON;	// This will bring us to SetState(E_LAMP_STATE.OP, E_LAMP_SUBSTATE.OP_WARMING)
	ELSE
		// Log event
		M_LogEventEnd('ON');

		nInternalEvent 		:= E_LAMP_EVENT.WARMED_UP;	// This will bring us to SetState(E_LAMP_STATE.OP, E_LAMP_SUBSTATE.OP_ON)
	END_IF
	
	M_SetStatus(E_LAMP_ERROR.OK);	

	RETURN;
END_IF

(* 
	if the timeout is detected before reaching the position, 
	then trigger the internal error event 
*)
toutCmd();
IF toutCmd.Q THEN
	// Log event
	M_LogEventError('ON command timed out');

	toutCmd(IN:=FALSE);	(* Reset Timer *)
	timer(IN:=FALSE);	(* Reset the signal duration timer *)
	
	nInternalEvent  := E_LAMP_EVENT.ERRTIMEOUTON;
	SetEvent(E_LAMP_EVENT.ERRTIMEOUTON);
	M_SetStatus(E_LAMP_ERROR.TIMEOUT_ON);	
END_IF
END_METHOD

METHOD ActivityWarmingUp
VAR_INPUT
END_VAR
(* 
	This activity waits for cfg.nWarmup seconds until the lamp has warmed up.
	It triggers E_LAMP_EVENT.WARMED_UP event. 
*)
SetAction('ActivityWarmingUp');

// Update the ON time
M_UpdateTimes(bOnState:=TRUE, bRestart:=FALSE, bReset:=FALSE);

(* 
	Warming is complete on expiration of the timer.
	If there is no warmup (cfg.nWarmup = 0), just set the event E_LAMP_EVENT.WARMED_UP.
*)
toutCmd();
IF toutCmd.Q OR cfg.nWarmup = 0 THEN
	// Log event
	M_LogEventEnd('ON');

	toutCmd(IN:=FALSE);	(* Reset Timer *)
	
	nInternalEvent 		:= E_LAMP_EVENT.WARMED_UP;	// This will bring us to (E_LAMP_STATE.OP, E_LAMP_SUBSTATE.OP_ON)
END_IF

// Check if the lamp has been ON longer than the time limit for that command.
IF stat.nTimeOnLimit > 0 AND stat.nTimeOn > stat.nTimeOnLimit THEN
	M_LogEventGeneral('Time ON limit reached during warmup. Switching lamp OFF.');
	nEvent  := E_LAMP_EVENT.LIMIT_ON;
	RETURN;
END_IF
END_METHOD

METHOD CheckForEvents
VAR_INPUT
END_VAR

(* 
	Start assuming the HW is OK. 
	This is needed to recover from the situation where 
	the HW was failing and now it is working.
*)
nEvent := E_LAMP_EVENT.HWOK;


(*
	Read all inputs, i.e. get status of INPUT signals based on ActiveLow configuration 
*)

bFault	:= M_GetLogicalState(i_bFault, cfg.bActiveLowFault) AND NOT cfg.bIgnoreFault;

(* The lamp ON feedback can be analog and/or digital. *)
stat.bOnDigital	:= M_GetLogicalState(i_bOn, cfg.bActiveLowOn);	// Digital feedback
stat.nOn		:= i_nOn;										// Analog  feedback

IF cfg.nAnalogThreshold <> 0	THEN
// Analog feedback is checked only if the threshold is not 0.0.
	stat.bOnAnalog	:=	((i_nOn > cfg.nAnalogThreshold) AND NOT cfg.bInvertAnalog) OR
						((i_nOn < cfg.nAnalogThreshold) AND     cfg.bInvertAnalog);
ELSE
	stat.bOnAnalog	:= FALSE;
END_IF
	
IF 	(stat.bOnDigital OR  stat.bOnAnalog)	THEN
	bOn	:= TRUE;
ELSE
	bOn	:= FALSE;
END_IF


M_UpdateTimes(bOnState:=bOn,bRestart:=FALSE, bReset:=FALSE);	// Update the Time


(* HW Status in textual form: 'ERROR', 'ON' or 'OFF' *)
IF 		bFault THEN
	stat.nHwStatus	:= E_LAMP_HW_STATUS.ERROR;
	stat.sHwStatus	:= 'ERROR';
ELSIF 	bOn   = TRUE  THEN
	stat.nHwStatus	:= E_LAMP_HW_STATUS.ON;
	stat.sHwStatus	:= 'ON';
ELSIF 	bOn   = FALSE  THEN
	stat.nHwStatus	:= E_LAMP_HW_STATUS.OFF;
	stat.sHwStatus	:= 'OFF';
END_IF

(* 
	Check for events in the following order: 
   	1) HW failure: without HW avilability there is no point to do anything
	2) Internal events: to allow completing the initiated commands before 
                        starting processing new commands. 
   	3) Commands: to react to external commands. Commands should be executed 
                 before processing HW signals to allow to start a recovery action.
   	4) HW signals:  such as Lamp is ON/OFF.
*)

IF 	i_nCouplerState <> 8 AND 
	NOT (ctrl.bExecute AND ctrl.nCommand = E_LAMP_COMMAND.RESET) THEN	
	// NOTE:	We give priority to RESET command in order 
	//			to be able to switch from OP to NOT_OP on RESET.
	(* Check if the HW is NOT OK *)
	(*
	If the hardware status is NOT OK, we cannot trust the readings.
	Variable i_nCouplerState has to be mapped to a State of a terminal, e.g. EK1100.
	The value should be 8.
 	*)
	SetEvent(E_LAMP_EVENT.ERRHW);
	M_SetStatus(E_LAMP_ERROR.HW_NOT_OP);

ELSIF nInternalEvent <> E_LAMP_EVENT.NONE THEN
	(* Handle internal events *)
	SetEvent(nInternalEvent);
	nInternalEvent := E_LAMP_EVENT.NONE;
ELSIF ctrl.bExecute = TRUE  THEN
	(* Handle commands *)
	ctrl.bExecute	:= FALSE;				(* Clear the Execute bit *)
	M_SetLastCommand(ctrl.nCommand);		(* Save the last command *)
	SetEvent(ctrl.nCommand);				(* Set the event *)
	ctrl.nCommand 	:= E_LAMP_COMMAND.NONE;	(* Clear the Command *)
ELSE
	(* Handle HW problems and unexpected bahaviour *)
	
	IF bFault THEN
		SetEvent(E_LAMP_EVENT.ERRFAULT);
		M_SetStatus(E_LAMP_ERROR.FAULT_SIG);
		RETURN;	
	END_IF

	IF stat.nSubstate = E_LAMP_SUBSTATE.NOTOP_READY_OFF OR 
	   stat.nSubstate = E_LAMP_SUBSTATE.NOTOP_READY_ON OR 
	   stat.nSubstate = E_LAMP_SUBSTATE.OP_DISABLING OR 
	   stat.nSubstate = E_LAMP_SUBSTATE.OP_OFF OR 
	   stat.nSubstate = E_LAMP_SUBSTATE.OP_ON	OR 
	   stat.nSubstate = E_LAMP_SUBSTATE.OP_ERROR THEN
	   
		(* Set events for ON and OFF *)		
		IF	bOn   = TRUE  THEN
			SetEvent(E_LAMP_EVENT.ISON);
		ELSIF	bOn   = FALSE THEN
			SetEvent(E_LAMP_EVENT.ISOFF);
		END_IF	
	END_IF	
(*
	IF stat.nSubstate = E_LAMP_SUBSTATE.OP_SWITCHING_ON THEN
		(* Set events for ON  *)		
		IF	bOn   = TRUE  THEN
			SetEvent(E_LAMP_EVENT.ISON);
		END_IF	
	END_IF	
	*)
END_IF
END_METHOD

METHOD M_GetRpcErrorText : STRING
VAR_INPUT
	ErrorCode:	INT;
END_VAR
VAR
	str:	STRING;
END_VAR
CASE ErrorCode OF
	E_LAMP_RPC_ERROR.OK:						str	:= 'OK';
	E_LAMP_RPC_ERROR.NOT_OP:					str	:= 'Cannot control lamp. Not in OP state.';
	E_LAMP_RPC_ERROR.NOT_NOTOP_READY:			str	:= 'Call failed. Not in NOTOP_READY.';
	E_LAMP_RPC_ERROR.NOT_NOTOP_NOTREADY:		str	:= 'Call failed. Not in NOTOP_NOTREADY/ERROR.';
	E_LAMP_RPC_ERROR.SWITCHING_ON:			str	:= 'Lamp OFF failed. Still switching ON.';
	E_LAMP_RPC_ERROR.SWITCHING_OFF:			str	:= 'Lamp ON failed. Still switching OFF.';
	E_LAMP_RPC_ERROR.COOLING:					str	:= 'Lamp ON failed. Still cooling down.';
	E_LAMP_RPC_ERROR.LOCAL:					str	:= 'RPC calls not allowed in Local mode.';
ELSE
	str	:= 'Unregistered RPC error.';
END_CASE

M_GetRpcErrorText	:= str;
END_METHOD

METHOD M_SetLastCommand
VAR_INPUT
	cmd:	E_LAMP_COMMAND;
END_VAR
stat.nLastCommand	:= cmd;

CASE cmd OF
	E_LAMP_COMMAND.RESET:
		stat.sLastCommand	:= 'RESET';
	E_LAMP_COMMAND.INIT:
		stat.sLastCommand	:= 'INIT';
	E_LAMP_COMMAND.STOP:
		stat.sLastCommand	:= 'STOP';
	E_LAMP_COMMAND.ENABLE:
		stat.sLastCommand	:= 'ENABLE';
	E_LAMP_COMMAND.DISABLE:
		stat.sLastCommand	:= 'DISABLE';
	E_LAMP_COMMAND.ON:
		stat.sLastCommand	:= 'ON';
	E_LAMP_COMMAND.OFF:
		stat.sLastCommand	:= 'OFF';
ELSE
		stat.sLastCommand	:= 'NONE';
END_CASE;
END_METHOD

METHOD M_SetRpcStatus : INT
VAR_INPUT
	nErrorCode:	E_LAMP_RPC_ERROR;
END_VAR
stat.nRpcErrorCode	:= nErrorCode;
stat.sRpcErrorText	:= M_GetRpcErrorText(nErrorCode);

M_SetRpcStatus		:= nErrorCode;
END_METHOD

METHOD M_UpdateCtrlParams : BOOL
VAR_INPUT
END_VAR
(* Turn the control signal ON  and set the intensity *)
q_bSwitch			:= M_GetLogicalState(TRUE, cfg.bActiveLowSwitch);
stat.lrIntensity	:= ctrl.lrIntensity;
q_nIntensity		:= LREAL_TO_INT(stat.lrIntensity / 100.0 * cfg.nFullRange);

// Save time limit for ON and clear it from the command parameters
stat.nTimeOnLimit	:= ctrl.nTimeOnLimit;
ctrl.nTimeOnLimit	:= 0;
END_METHOD

{attribute 'TcRpcEnable':='1'}
METHOD RPC_Disable : INT
VAR_INPUT
END_VAR
// RPC calls are not allowed in Local mode.
IF stat.bLocal THEN
	RPC_Disable	:= M_SetRpcStatus(E_LAMP_RPC_ERROR.LOCAL);
	RETURN;
END_IF

// Disable command is accepted only if device is in OP state.
IF stat.nState <> E_LAMP_STATE.OP THEN
	RPC_Disable	:= M_SetRpcStatus(E_LAMP_RPC_ERROR.NOT_OP);
	RETURN;
ELSE
	// Set disable command
	ctrl.nCommand := E_LAMP_COMMAND.DISABLE;
	ctrl.bExecute := TRUE;
	
	// Call was successful
	RPC_Disable	:= M_SetRpcStatus(E_LAMP_RPC_ERROR.OK);
END_IF
END_METHOD

{attribute 'TcRpcEnable':='1'}
METHOD RPC_Enable : INT
VAR_INPUT
END_VAR
// RPC calls are not allowed in Local mode.
IF stat.bLocal THEN
	RPC_Enable	:= M_SetRpcStatus(E_LAMP_RPC_ERROR.LOCAL);
	RETURN;
END_IF

// Enable command is accepted only if device is in NOTOP_READY.
IF	stat.nState = E_LAMP_STATE.NOTOP					AND  
	stat.nSubstate <> E_LAMP_SUBSTATE.NOTOP_READY_OFF	AND  
	stat.nSubstate <> E_LAMP_SUBSTATE.NOTOP_READY_ON		THEN
	RPC_Enable	:= M_SetRpcStatus(E_LAMP_RPC_ERROR.NOT_NOTOP_READY);
	RETURN;
ELSE
	// Set enable command
	ctrl.nCommand := E_LAMP_COMMAND.ENABLE;
	ctrl.bExecute := TRUE;
	
	// Call was successful
	RPC_Enable	:= M_SetRpcStatus(E_LAMP_RPC_ERROR.OK);
END_IF
END_METHOD

{attribute 'TcRpcEnable':='1'}
METHOD RPC_Init : INT
VAR_INPUT
END_VAR
IF stat.bLocal THEN
	// RPC calls are not allowed in Local mode.
	RPC_Init	:= M_SetRpcStatus(E_LAMP_RPC_ERROR.LOCAL);
	RETURN;
ELSIF i_nCouplerState <> 8 THEN
	// EtherCAT is not OPERATIONAL, device cannot be initialised.
	RPC_Init	:= M_SetRpcStatus(E_LAMP_RPC_ERROR.NOT_OP);
	RETURN;
ELSIF	stat.nSubstate <> E_LAMP_SUBSTATE.NOTOP_NOTREADY	AND  
		stat.nSubstate <> E_LAMP_SUBSTATE.NOTOP_ERROR		THEN
	// Init command is accepted only if device is in NOTOP_NOTREADY or ERROR.
	RPC_Init	:= M_SetRpcStatus(E_LAMP_RPC_ERROR.NOT_NOTOP_NOTREADY);
	RETURN;
ELSE
	// Set INIT command
	ctrl.nCommand := E_LAMP_COMMAND.INIT;
	ctrl.bExecute := TRUE;
	
	// Call was successful
	RPC_Init	:= M_SetRpcStatus(E_LAMP_RPC_ERROR.OK);
END_IF
END_METHOD

{attribute 'TcRpcEnable':='1'}
METHOD RPC_Off : INT
VAR_INPUT
END_VAR
// RPC calls are not allowed in Local mode.
IF stat.bLocal THEN
	RPC_Off	:= M_SetRpcStatus(E_LAMP_RPC_ERROR.LOCAL);
	RETURN;
END_IF

// OFF command is accepted only in OP state.
IF	stat.nState <> E_LAMP_STATE.OP	THEN
	RPC_Off	:= M_SetRpcStatus(E_LAMP_RPC_ERROR.NOT_OP);
	RETURN;
ELSIF stat.nSubstate = E_LAMP_SUBSTATE.OP_SWITCHING_ON THEN
	// Lamp should not be commanded to go OFF if being switched ON.
	RPC_Off	:= M_SetRpcStatus(E_LAMP_RPC_ERROR.SWITCHING_ON);
	RETURN;
ELSE
	// Set OFF command
	ctrl.nCommand := E_LAMP_COMMAND.OFF;
	ctrl.bExecute := TRUE;
	
	// Call was successful
	RPC_Off	:= M_SetRpcStatus(E_LAMP_RPC_ERROR.OK);
END_IF
END_METHOD

{attribute 'TcRpcEnable':='1'}
METHOD RPC_On : INT
VAR_INPUT
	in_lrIntensity:		LREAL	:= 0.0;	// Intensity 0-100% [%]
	in_nTimeOnLimit:	UDINT	:= 0;	// Auto OFF after this time [sec]. 0 - no limit
END_VAR
// RPC calls are not allowed in Local mode.
IF stat.bLocal THEN
	RPC_On	:= M_SetRpcStatus(E_LAMP_RPC_ERROR.LOCAL);
	RETURN;
END_IF

// ON command is accepted only in OP state and NOT COOLING.
IF	stat.nState <> E_LAMP_STATE.OP	THEN
	RPC_On	:= M_SetRpcStatus(E_LAMP_RPC_ERROR.NOT_OP);
	RETURN;
ELSIF stat.nSubstate = E_LAMP_SUBSTATE.OP_COOLING THEN
	RPC_On	:= M_SetRpcStatus(E_LAMP_RPC_ERROR.COOLING);
	RETURN;
ELSIF stat.nSubstate = E_LAMP_SUBSTATE.OP_SWITCHING_OFF THEN
	// Lamp should not be commanded to go ON if being switched OFF.
	RPC_On	:= M_SetRpcStatus(E_LAMP_RPC_ERROR.SWITCHING_OFF);
	RETURN;
ELSE
	// Set ON command
	ctrl.nCommand 		:= E_LAMP_COMMAND.ON;
	ctrl.lrIntensity	:= in_lrIntensity;
	ctrl.nTimeOnLimit	:= in_nTimeOnLimit;
	ctrl.bExecute 		:= TRUE;
	
	// Call was successful
	RPC_On	:= M_SetRpcStatus(E_LAMP_RPC_ERROR.OK);
END_IF
END_METHOD

{attribute 'TcRpcEnable':='1'}
METHOD RPC_Reset : INT
VAR_INPUT
END_VAR
// RPC calls are not allowed in Local mode.
IF stat.bLocal THEN
	RPC_Reset	:= M_SetRpcStatus(E_LAMP_RPC_ERROR.LOCAL);
	RETURN;
END_IF

ctrl.nCommand := E_LAMP_COMMAND.RESET;
ctrl.bExecute := TRUE;

// Call was successful
RPC_Reset	:= M_SetRpcStatus(E_LAMP_RPC_ERROR.OK);
END_METHOD

{attribute 'TcRpcEnable':='1'}
METHOD RPC_SetDebug : INT
VAR_INPUT
	in_bDebug:	BOOL 	:= FALSE;		// If TRUE, activate event logging of Debug type
END_VAR
// Enable/disable Debugging
cfg.bDebug	:= in_bDebug;

// Call was successful
RPC_SetDebug	:= M_SetRpcStatus(E_LAMP_RPC_ERROR.OK);
END_METHOD

{attribute 'TcRpcEnable':='1'}
METHOD RPC_SetLog : INT
VAR_INPUT
	in_bLog:	BOOL 	:= FALSE;		// If TRUE, activate event logging
END_VAR
// Enable/disable Logging
cfg.bLog	:= in_bLog;

// Call was successful
RPC_SetLog	:= M_SetRpcStatus(E_LAMP_RPC_ERROR.OK);
END_METHOD

{attribute 'TcRpcEnable':='1'}
METHOD RPC_Stop : INT
VAR_INPUT
END_VAR
// RPC calls are not allowed in Local mode.
IF stat.bLocal THEN
	RPC_Stop	:= M_SetRpcStatus(E_LAMP_RPC_ERROR.LOCAL);
	RETURN;
END_IF

ctrl.nCommand := E_LAMP_COMMAND.STOP;
ctrl.bExecute := TRUE;

// Call was successful
RPC_Stop	:= M_SetRpcStatus(E_LAMP_RPC_ERROR.OK);
END_METHOD

END_FUNCTION_BLOCK

// ---- POUs/FB_LAMP_BASE.TcPOU
FUNCTION_BLOCK FB_LAMP_BASE
VAR_INPUT
	{attribute 'OPC.UA.DA':='0'}
	in_sName:				STRING	:= 'Lamp';	// Instance name
	{attribute 'OPC.UA.DA':='0'}
	in_bActiveLowFault:		BOOL 	:= FALSE;	(* If TRUE, Fault signal is Active Low *)
	{attribute 'OPC.UA.DA':='0'}
	in_bActiveLowOn:		BOOL 	:= FALSE;	(* If TRUE, On signal is Active Low *)
	{attribute 'OPC.UA.DA':='0'}
	in_bActiveLowSwitch:	BOOL 	:= FALSE;	(* If TRUE, Switch ctrl signal is Active Low *)

	{attribute 'OPC.UA.DA':='0'}
	in_bIgnoreFault:		BOOL 	:= FALSE;	(* If TRUE, Fault feedback signal is ignored *)
	{attribute 'OPC.UA.DA':='0'}
	in_bInitialState:		BOOL 	:= FALSE;	(* default lamp state is OFF *)
	{attribute 'OPC.UA.DA':='0'}
	in_bInvertAnalog:		BOOL 	:= FALSE;	(* If TRUE, analog feedback is active, if signal < nAnalogThreshold *)
	
	{attribute 'OPC.UA.DA':='0'}
	in_lrInitialIntensity:	LREAL 	:= 0.0;		// Initial intensity [%]. Default 0.0.
	
	{attribute 'OPC.UA.DA':='0'}
	in_nAnalogThreshold:	INT 	:= 0;		(* Analog feedback signal threshold [bits].
										   		If this signal is used, any value above it will indicate that the lamp is ON. *)
	{attribute 'OPC.UA.DA':='0'}
	in_nFullRange:			UDINT 	:= 32767;	(* Full range of A/D converter for analog output for intensity control. Default is 15-bit.
										   		Beckhoff 16-bit analog output terminals include the sign.
										   		Effectively, for 0-10V terminals, this is a 15-bit resolution.  *)
	{attribute 'OPC.UA.DA':='0'}
	in_nSigStablePeriod:	UDINT 	:= 100;		(* signal is stable if it has been constant for so long [msec] *)
	{attribute 'OPC.UA.DA':='0'}
	in_nTimeout:     		UDINT 	:= 3000;	(* timeout for transitions [msec] *)

	{attribute 'OPC.UA.DA':='0'}
	in_nCooldown:			UDINT 	:= 0;		(* Cooldown time [sec] *)
	{attribute 'OPC.UA.DA':='0'}
	in_nMaxOn:				UDINT 	:= 0;		(* Maximum time for lamp to be ON [sec]. Zero means no limit. *)
	{attribute 'OPC.UA.DA':='0'}
	in_nWarmup:				UDINT 	:= 0;		(* Warmup time [sec] *)

	{attribute 'OPC.UA.DA':='0'}
	in_bLogExtTime:			BOOL 	:= FALSE;		// If TRUE, use external time in event logs. Default FALSE.
	{attribute 'OPC.UA.DA':='0'}
	in_bLog:				BOOL 	:= TRUE;		// If TRUE, log events. Default TRUE.
END_VAR
VAR_OUTPUT
END_VAR
VAR RETAIN
END_VAR
VAR
	{attribute 'OPC.UA.DA' := '1'}
	cfg:		T_LAMP_CFG;	
	{attribute 'OPC.UA.DA' := '1'}
	ctrl:		T_LAMP_CTRL;	
	{attribute 'OPC.UA.DA' := '1'}
	{attribute 'OPC.UA.DA.Access' := '1'}
	info:		T_LAMP_INFO;	(* ReadOnly *)
	{attribute 'OPC.UA.DA' := '1'}
	{attribute 'OPC.UA.DA.Access' := '1'}
	stat:		T_LAMP_STAT;	(* ReadOnly *)

	{attribute 'OPC.UA.DA' := '0'}
	nEvent:		      	DINT := E_LAMP_EVENT.NONE;
	{attribute 'OPC.UA.DA' := '0'}
	nInternalEvent:		DINT := E_LAMP_EVENT.NONE;
	
	// Operational Events
	{attribute 'OPC.UA.DA' := '0'}
	fbEventStart:	FB_TcMessage;
	{attribute 'OPC.UA.DA' := '0'}
	fbEventEnd:		FB_TcMessage;
	{attribute 'OPC.UA.DA' := '0'}
	fbEventError:	FB_TcMessage;
	{attribute 'OPC.UA.DA' := '0'}
	fbEventDebug:	FB_TcMessage;
	{attribute 'OPC.UA.DA' := '0'}
	fbEventGeneral:	FB_TcMessage;
	
	(***** Physical signals - to be mapped!!! *****)

	(* Outputs *)

	(* Inputs *)
	
	// Flag if the device is ready to receive commands.
	// It takes a couple of cycles for the system to read inputs after reboot.
	{attribute 'OPC.UA.DA' := '0'}
	bDeviceReady:	BOOL 	:= FALSE;

END_VAR

// On first cycle configure from input params and internally execute M_UserConfigure()
IF NOT bDeviceReady THEN
	// Set device Configuration
	M_Configure();
	RETURN;
END_IF

// Increment counter.
// This will be seen as 'alive' flag.
stat.nCycleCounter	:= stat.nCycleCounter + 1;


(* === Check for commands and internal events to be processed === *)
CheckForEvents();

(* === Process events according to the State Machine === *)
ProcessEvents();

METHOD ActionDisableExecute
VAR_INPUT
END_VAR
END_METHOD

METHOD ActionEnableComplete
VAR_INPUT
END_VAR
END_METHOD

METHOD ActionEnableExecute
VAR_INPUT
END_VAR
END_METHOD

METHOD ActionErrExecute
VAR
END_VAR
END_METHOD

METHOD ActionInitAbort
VAR_INPUT
END_VAR
END_METHOD

METHOD ActionInitComplete
VAR_INPUT
END_VAR
END_METHOD

METHOD ActionInitExecute
VAR_INPUT
END_VAR
END_METHOD

METHOD ActionInitReject
VAR_INPUT
END_VAR
END_METHOD

METHOD ActionMaxOnFailure
VAR_INPUT
END_VAR
END_METHOD

METHOD ActionOffExecute
VAR_INPUT
END_VAR
END_METHOD

METHOD ActionOnExecute
VAR_INPUT
END_VAR
END_METHOD

METHOD ActionResetExecute
VAR_INPUT
END_VAR
END_METHOD

METHOD ActionUnexpExecute
VAR
END_VAR
END_METHOD

METHOD ActivityCoolingDown
VAR_INPUT
END_VAR
END_METHOD

METHOD ActivityDisabling
VAR_INPUT
END_VAR
END_METHOD

METHOD ActivityInitializing
VAR_INPUT
END_VAR
END_METHOD

METHOD ActivityOff
VAR_INPUT
END_VAR
END_METHOD

METHOD ActivityOn
VAR_INPUT
END_VAR
END_METHOD

METHOD ActivitySwitchingOff
VAR_INPUT
END_VAR
END_METHOD

METHOD ActivitySwitchingOn
VAR_INPUT
END_VAR
END_METHOD

METHOD ActivityWarmingUp
VAR_INPUT
END_VAR
END_METHOD

METHOD CheckForEvents
VAR_INPUT
END_VAR
END_METHOD

METHOD M_CheckTimeLeft
VAR_INPUT
END_VAR
VAR
	nTimeLeft:	UDINT 	:= 0;
	nTimeLimit:	UDINT 	:= 0;
	bCheck:		BOOL	:= TRUE;
END_VAR
IF 	stat.nSubstate = E_LAMP_SUBSTATE.OP_ON  OR 
	stat.nSubstate = E_LAMP_SUBSTATE.OP_WARMING  THEN
	IF cfg.nMaxOn > 0  AND  stat.nTimeOnLimit > 0 THEN
		nTimeLimit	:= MIN (cfg.nMaxOn, stat.nTimeOnLimit);
	ELSIF cfg.nMaxOn > 0  THEN
		nTimeLimit	:= cfg.nMaxOn;
	ELSIF stat.nTimeOnLimit > 0 THEN
		nTimeLimit	:= stat.nTimeOnLimit;
	END_IF	

	IF nTimeLimit > 0 THEN
		nTimeLeft	:= nTimeLimit - stat.nTimeOn;
	ELSE
		nTimeLeft	:= 0;
		bCheck		:= FALSE;
	END_IF	
ELSE
	// Lamp is not ON, remaining time is zero.
	nTimeLeft	:= 0;
	bCheck		:= FALSE;
END_IF

stat.nTimeLeft		:= nTimeLeft;
stat.bCheckTimeLeft	:= bCheck;
END_METHOD

METHOD M_Configure : BOOL
VAR_INPUT
END_VAR
VAR
     fbGetCurTaskIdx:	GETCURTASKINDEX;
END_VAR
// If device is ready, there is nothing to configure.
IF bDeviceReady THEN
	RETURN;
END_IF

// If first cycle, copy configuration AND RETURN in order for the system to read all inputs before doing any work
IF stat.nCycleCounter = 0 THEN
	cfg.sName				:=	in_sName;			// Instance name

	cfg.bActiveLowFault		:= in_bActiveLowFault;	(* If TRUE, Fault signal is Active Low *)
	cfg.bActiveLowOn		:= in_bActiveLowOn;		(* If TRUE, On signal is Active Low *)
	cfg.bActiveLowSwitch	:= in_bActiveLowSwitch;	(* If TRUE, Switch ctrl signal is Active Low *)

	cfg.bIgnoreFault		:= in_bIgnoreFault;		(* If TRUE, Fault feedback signal is ignored *)
	cfg.bInitialState		:= in_bInitialState;	(* default lamp state is OFF *)
	cfg.bInvertAnalog		:= in_bInvertAnalog;	(* If TRUE, analog feedback is active, if signal < nAnalogThreshold *)
	
	cfg.lrInitialIntensity	:= in_lrInitialIntensity;	// Initial intensity [%]. Default 0.0.
	// If the initial state is OFF, set intensity to zero.
	IF NOT cfg.bInitialState THEN
		cfg.lrInitialIntensity	:= 0.0;
	END_IF

	cfg.nAnalogThreshold	:= in_nAnalogThreshold;	(* Analog feedback signal threshold [bits].
										   			If this signal is used, any value above it will indicate that the lamp is ON. *)
	cfg.nFullRange			:= in_nFullRange;		(* Full range of A/D converter for analog output for intensity control. Default is 15-bit.
										   			Beckhoff 16-bit analog output terminals include the sign.
										   			Effectively, for 0-10V terminals, this is a 15-bit resolution.  *)
	cfg.nSigStablePeriod	:= in_nSigStablePeriod;	(* signal is stable if it has been constant for so long [msec] *)
	cfg.nTimeout			:= in_nTimeout;			(* timeout for transitions [msec] *)


	cfg.nCooldown			:= in_nCooldown;		(* Cooldown time [sec] *)
	cfg.nMaxOn				:= in_nMaxOn;			(* Maximum time for lamp to be ON [sec] *)
	cfg.nWarmup				:= in_nWarmup;			(* Warmup time [sec] *)

	cfg.bLogExtTime			:= in_bLogExtTime;		// If TRUE, use external time in event logs
	cfg.bLog				:= in_bLog;				// If TRUE, use external time in event logs

	// Get the version number 
	stat.sLibVersion	:= stLibVersion_ESO_LDC_Lamp_Library.sVersion;

	// Get cycle time in microsec.
	// CycleTime in _TaskInfo is given in 100 ns. 1 us = 1000 ns
	fbGetCurTaskIdx();
	stat.nCycleTime	:=  (TwinCAT_SystemInfoVarList._TaskInfo[fbGetCurTaskIdx.index].CycleTime)/10;
	
	// Increment counter.
	stat.nCycleCounter	:= stat.nCycleCounter + 1;
	RETURN;
ELSIF (stat.nCycleCounter * stat.nCycleTime) < 5000000 THEN
	// EtherCAT is normally ready after 3.5 sec.
	// We give it 5 sec to consider it to be ready.
	// Increment counter.
	stat.nCycleCounter	:= stat.nCycleCounter + 1;
	RETURN;
END_IF

// The system shoud be ready, i.e. coupler state is 8.

// Create Event instances
fbEventStart.CreateEx	(TC_EVENTS.LampOpsEventClass.ActionStart,0);
fbEventEnd.CreateEx		(TC_EVENTS.LampOpsEventClass.ActionEnd,0);
fbEventError.CreateEx	(TC_EVENTS.LampOpsEventClass.Error,0);
fbEventDebug.CreateEx	(TC_EVENTS.LampOpsEventClass.Debug,0);
fbEventGeneral.CreateEx	(TC_EVENTS.LampOpsEventClass.General,0);

// The device is ready now.
bDeviceReady := TRUE;


// Clear errors
M_SetStatus(E_LAMP_ERROR.OK);
END_METHOD

METHOD M_GetErrorText : STRING
VAR_INPUT
	ErrorCode:	DINT;
END_VAR
VAR
	sErrorText:	STRING;
END_VAR
CASE ErrorCode OF
	E_LAMP_ERROR.OK:					sErrorText	:= 'OK';
	E_LAMP_ERROR.HW_NOT_OP:			sErrorText	:= 'ERROR: TwinCAT not in OP state or CouplerState not mapped.';
	E_LAMP_ERROR.INIT_FAILURE:		sErrorText	:= 'ERROR: INIT command aborted due to STOP or RESET.';
	E_LAMP_ERROR.UNEXPECTED_OFF:		sErrorText	:= 'ERROR: Lamp unexpectedly switched OFF.';
	E_LAMP_ERROR.UNEXPECTED_ON:		sErrorText	:= 'ERROR: Lamp unexpectedly switched ON.';
	E_LAMP_ERROR.FAULT_SIG:			sErrorText	:= 'ERROR: Fault signal active.';
	E_LAMP_ERROR.MAXON:				sErrorText	:= 'ERROR: Lamp maximum ON time exceeded.';
	E_LAMP_ERROR.STILL_COOLING:		sErrorText	:= 'ERROR: ON command not allowed while cooling.';
	E_LAMP_ERROR.TIMEOUT_DISABLE:		sErrorText	:= 'ERROR: Disable timed out.';
	E_LAMP_ERROR.TIMEOUT_INIT:		sErrorText	:= 'ERROR: Init timed out.';
	E_LAMP_ERROR.TIMEOUT_OFF:			sErrorText	:= 'ERROR: Switching OFF timed out.';
	E_LAMP_ERROR.TIMEOUT_ON:			sErrorText	:= 'ERROR: Switching ON timed out.';
	E_LAMP_ERROR.SIM_NOT_INITIALISED:	sErrorText	:= 'ERROR: Lamp simulator not initialised.';
	E_LAMP_ERROR.SIM_NULL_POINTER:	sErrorText	:= 'ERROR: NULL pointer to Lamp.';
ELSE
	sErrorText	:= 'Unregistered error.';
END_CASE

M_GetErrorText	:= sErrorText;
END_METHOD

METHOD M_GetLogicalState : BOOL
(*
	This method returns the state of the variable based on its 
	activeLow configuration.
	Syntax:
		bState	:= M_GetLogicalState (<var value>,  <activeLow cfg>);
		
	Example 1:
		var = TRUE;
		activeLow = FALSE;
		bState	:= M_GetLogicalState (TRUE,  FALSE); = TRUE

	Example 2:
		var = TRUE;
		activeLow = TRUE;
		bState	:= M_GetLogicalState (TRUE,  TRUE); = FALSE
*)
VAR_INPUT
	state:		BOOL;
	activeLow:	BOOL;
END_VAR
IF activeLow THEN
	M_GetLogicalState := NOT state;
ELSE
	M_GetLogicalState := state;
END_IF
END_METHOD

(*
	This method returns absolute time rounded to seconds.
*)
METHOD M_GetTimeInSec : UDINT
VAR_INPUT
END_VAR
VAR
END_VAR
// System time is given in 100ns. Divide by 10000000 to get in seconds. 
M_GetTimeInSec	:= ULINT_TO_UDINT(Tc2_System.F_GetSystemTime() / 10000000);
END_METHOD

METHOD M_LogEventDebug : BOOL
VAR_INPUT
	sText:	STRING	:= '';
END_VAR
// Log Debug events only if both logging and debugging is enabled
IF  cfg.bLog AND cfg.bDebug THEN
	fbEventDebug.ipArguments.Clear().AddString(sText);
	fbEventDebug.Send(0);
END_IF
END_METHOD

METHOD M_LogEventEnd : BOOL
VAR_INPUT
	sText:	STRING	:= '';
END_VAR
// Log only if logging is enabled
IF  NOT cfg.bLog THEN
	RETURN;
END_IF

fbEventEnd.ipArguments.Clear().AddString(sText);
fbEventEnd.Send(0);
END_METHOD

METHOD M_LogEventError : BOOL
VAR_INPUT
	sText:	STRING	:= '';
END_VAR
// Log only if logging is enabled
IF  NOT cfg.bLog THEN
	RETURN;
END_IF

fbEventError.ipArguments.Clear().AddString(sText);
fbEventError.Send(0);
END_METHOD

METHOD M_LogEventGeneral : BOOL
VAR_INPUT
	sText:	STRING	:= '';
END_VAR
// Log only if logging is enabled
IF  NOT cfg.bLog THEN
	RETURN;
END_IF

fbEventGeneral.ipArguments.Clear().AddString(sText);
fbEventGeneral.Send(0);
END_METHOD

METHOD M_LogEventStart : BOOL
VAR_INPUT
	sText:	STRING	:= '';
END_VAR
// Log only if logging is enabled
IF  NOT cfg.bLog THEN
	RETURN;
END_IF

fbEventStart.ipArguments.Clear().AddString(sText);
fbEventStart.Send(0);
END_METHOD

METHOD M_SetStatus
VAR_INPUT
	nErrorCode:	E_LAMP_ERROR;
END_VAR
stat.nErrorCode 	:= nErrorCode;
stat.sErrorText 	:= M_GetErrorText(nErrorCode);

IF nErrorCode <> E_LAMP_ERROR.OK THEN
	stat.sStatus	:= 'ERROR';
	stat.nStatus	:= E_LAMP_STATUS.ERROR;
ELSE
	stat.sStatus	:= 'OK';
	stat.nStatus	:= E_LAMP_STATUS.OK;
END_IF
END_METHOD

METHOD M_UpdateCtrlParams : BOOL
VAR_INPUT
END_VAR
END_METHOD

METHOD M_UpdateTimes
VAR_INPUT
	bOnState:	BOOL;	// State of ON status signal
	bRestart:	BOOL := FALSE;	// If TRUE, restart ON time after new command
	bReset:		BOOL := FALSE;	// If TRUE, reset ON /OFF times
END_VAR
VAR
	nCurrentTime:	UDINT;
END_VAR
nCurrentTime	:= M_GetTimeInSec();

IF bReset OR stat.nSubstate = E_LAMP_SUBSTATE.NOTOP_NOTREADY THEN
	stat.nTimeOnStart		:= nCurrentTime;
	stat.nTimeOnTotalStart	:= nCurrentTime;
	stat.nTimeOffStart		:= nCurrentTime;
	stat.nTimeOnTotal		:= 0;
	stat.nTimeOn			:= 0;
	stat.nTimeOff			:= 0;
	RETURN;
END_IF


IF bOnState THEN
	// Lamp state is ON.
	// In order to avoid OFF time jumps, reset OFF start time.
	stat.nTimeOffStart	:= nCurrentTime;
	
	// Check if the lamp has already been ON.
	IF	stat.nSubstate = E_LAMP_SUBSTATE.OP_ON OR
		stat.nSubstate = E_LAMP_SUBSTATE.OP_WARMING THEN
		// Lamp has already been ON
		stat.nTimeOnTotal	:= nCurrentTime - stat.nTimeOnTotalStart;

		IF bRestart THEN
			stat.nTimeOnStart	:= nCurrentTime;
			stat.nTimeOn		:= 0;
		ELSE
			stat.nTimeOn		:= nCurrentTime - stat.nTimeOnStart;
		END_IF
	ELSE
		// Lamp has been OFF
		stat.nTimeOnStart		:= nCurrentTime;
		stat.nTimeOnTotalStart	:= nCurrentTime;
		stat.nTimeOnTotal		:= 0;
		stat.nTimeOn			:= 0;
		stat.nTimeOff			:= 0;
	END_IF

	// Check if the lamp has been ON for too long, i.e. cfg.nMaxOn exceeded.
	IF stat.nTimeOn > cfg.nMaxOn AND cfg.nMaxOn > 0 THEN
		nInternalEvent  := E_LAMP_EVENT.ERRMAXON;
		RETURN;
	END_IF

ELSE
	// Lamp state is OFF.
	// In order to avoid OFF time jumps, reset OFF start time.
	stat.nTimeOnStart	:= nCurrentTime;
	
	// Check if the lamp has already been OFF.
	IF 	stat.nSubstate = E_LAMP_SUBSTATE.OP_OFF OR
		stat.nSubstate = E_LAMP_SUBSTATE.OP_COOLING THEN
		// Lamp has already been OFF
		stat.nTimeOff	:= nCurrentTime - stat.nTimeOffStart;
	ELSE
		IF bRestart THEN
			stat.nTimeOffStart	:= nCurrentTime;
			stat.nTimeOff		:= 0;
		ELSE
			stat.nTimeOff		:= nCurrentTime - stat.nTimeOffStart;
		END_IF
	END_IF
END_IF
END_METHOD

METHOD ProcessEvents
VAR_INPUT
END_VAR

VAR
END_VAR

(* 
	Before processing the event, execute the Do-Activity tasks. 
	Note that, in case of orthogonal regions, more than one Do-Activity 
	could run in the same PLC cycle.
	Note: Most of these activities have timeouts since they take time.
*)

IF stat.nSubstate = E_LAMP_SUBSTATE.NOTOP_INITIALIZING THEN
	ActivityInitializing();
END_IF

IF stat.nSubstate = E_LAMP_SUBSTATE.OP_SWITCHING_ON THEN
	ActivitySwitchingOn();
END_IF

IF stat.nSubstate = E_LAMP_SUBSTATE.OP_ON THEN
	ActivityOn();	// Just update times
END_IF

IF stat.nSubstate = E_LAMP_SUBSTATE.OP_WARMING THEN
	ActivityWarmingUp();
END_IF

IF stat.nSubstate = E_LAMP_SUBSTATE.OP_SWITCHING_OFF THEN
	ActivitySwitchingOff();
END_IF

IF stat.nSubstate = E_LAMP_SUBSTATE.OP_COOLING THEN
	ActivityCoolingDown();
END_IF

IF stat.nSubstate = E_LAMP_SUBSTATE.OP_OFF THEN
	ActivityOff();	// Just update times
END_IF

IF stat.nSubstate = E_LAMP_SUBSTATE.OP_DISABLING THEN
	ActivityDisabling();
END_IF


//
// Check remaining time 
//
M_CheckTimeLeft();


(* 
	Evaluate state machine transitions.
*)

CASE stat.nState OF

//***********************************
// NOTOP
//***********************************
E_LAMP_STATE.NOTOP:

	(* Transitions from NOTOP substates *)
	CASE stat.nSubstate OF
	
	E_LAMP_SUBSTATE.NOTOP_NOTREADY:		
		IF nEvent = E_LAMP_EVENT.RESET THEN
			ActionResetExecute();
			SetState(E_LAMP_STATE.NOTOP, E_LAMP_SUBSTATE.NOTOP_NOTREADY);
			RETURN;
		ELSIF nEvent = E_LAMP_EVENT.INIT THEN
			ActionInitExecute();
			SetState(E_LAMP_STATE.NOTOP, E_LAMP_SUBSTATE.NOTOP_INITIALIZING);
			RETURN;
		END_IF
		
	E_LAMP_SUBSTATE.NOTOP_INITIALIZING:			
		IF nEvent = E_LAMP_EVENT.RESET THEN
			ActionInitAbort();
			SetState(E_LAMP_STATE.NOTOP, E_LAMP_SUBSTATE.NOTOP_NOTREADY);
			RETURN;
		ELSIF nEvent = E_LAMP_EVENT.STOP THEN
			ActionInitAbort();
			SetState(E_LAMP_STATE.NOTOP, E_LAMP_SUBSTATE.NOTOP_NOTREADY);
			RETURN;
		ELSIF nEvent = E_LAMP_EVENT.ERRINIT THEN
			SetState(E_LAMP_STATE.NOTOP, E_LAMP_SUBSTATE.NOTOP_NOTREADY);
			RETURN;
		ELSIF nEvent = E_LAMP_EVENT.INITOFF THEN
			ActionInitComplete();
			SetState(E_LAMP_STATE.NOTOP, E_LAMP_SUBSTATE.NOTOP_READY_OFF);
			RETURN;
		ELSIF nEvent = E_LAMP_EVENT.INITON THEN
			ActionInitComplete();
			SetState(E_LAMP_STATE.NOTOP, E_LAMP_SUBSTATE.NOTOP_READY_ON);
			RETURN;
		END_IF
		
	E_LAMP_SUBSTATE.NOTOP_READY_OFF:			
		IF nEvent = E_LAMP_EVENT.RESET THEN
			ActionResetExecute();
			SetState(E_LAMP_STATE.NOTOP, E_LAMP_SUBSTATE.NOTOP_NOTREADY);
			RETURN;
		ELSIF nEvent = E_LAMP_EVENT.ISON THEN
			ActionUnexpExecute();
			SetState(E_LAMP_STATE.NOTOP, E_LAMP_SUBSTATE.NOTOP_READY_ON);
			RETURN;
		ELSIF nEvent = E_LAMP_EVENT.ENABLE THEN
			ActionEnableComplete();
			SetState(E_LAMP_STATE.OP, E_LAMP_SUBSTATE.OP_OFF);
			RETURN;
		END_IF

	E_LAMP_SUBSTATE.NOTOP_READY_ON:			
		IF nEvent = E_LAMP_EVENT.RESET THEN
			ActionResetExecute();
			SetState(E_LAMP_STATE.NOTOP, E_LAMP_SUBSTATE.NOTOP_NOTREADY);
			RETURN;
		ELSIF nEvent = E_LAMP_EVENT.ISOFF THEN
			ActionUnexpExecute();
			SetState(E_LAMP_STATE.NOTOP, E_LAMP_SUBSTATE.NOTOP_READY_OFF);
			RETURN;
		ELSIF nEvent = E_LAMP_EVENT.ENABLE THEN
			ActionEnableComplete();
			SetState(E_LAMP_STATE.OP, E_LAMP_SUBSTATE.OP_ON);
			RETURN;
		END_IF

	E_LAMP_SUBSTATE.NOTOP_ERROR:			
		IF nEvent = E_LAMP_EVENT.HWOK THEN
			SetState(E_LAMP_STATE.NOTOP, E_LAMP_SUBSTATE.NOTOP_NOTREADY);
			RETURN;
		END_IF
		
	END_CASE

	(* Transitions from any NOTOP substate *)
	IF nEvent = E_LAMP_EVENT.ERRHW THEN
		SetState(E_LAMP_STATE.NOTOP, E_LAMP_SUBSTATE.NOTOP_ERROR);
		RETURN;
	ELSIF nEvent = E_LAMP_EVENT.ERRFAULT THEN
		SetState(E_LAMP_STATE.NOTOP, E_LAMP_SUBSTATE.NOTOP_ERROR);			
		RETURN;
	END_IF
	
//***********************************
// OPERATIONAL
//***********************************
E_LAMP_STATE.OP:

	(* Transitions from OP substates *)
	CASE stat.nSubstate OF
	E_LAMP_SUBSTATE.OP_OFF:			
		IF nEvent = E_LAMP_EVENT.ON THEN
			ActionOnExecute();
			SetState(E_LAMP_STATE.OP, E_LAMP_SUBSTATE.OP_SWITCHING_ON);
			RETURN;
		ELSIF nEvent = E_LAMP_EVENT.OFF THEN
			// Nothing to do. Just clear previous error, if any.
			M_SetStatus(E_LAMP_ERROR.OK);
			RETURN;
		ELSIF nEvent = E_LAMP_EVENT.ISON THEN
			ActionUnexpExecute();
			SetState(E_LAMP_STATE.OP, E_LAMP_SUBSTATE.OP_ON);
			RETURN;
		ELSIF nEvent = E_LAMP_EVENT.DISABLE THEN
			ActionDisableExecute();
			SetState(E_LAMP_STATE.OP, E_LAMP_SUBSTATE.OP_DISABLING);
			RETURN;		
		END_IF

	E_LAMP_SUBSTATE.OP_SWITCHING_ON:			
		IF nEvent = E_LAMP_EVENT.ISON THEN
			// This event will happen if there is warmup
			SetState(E_LAMP_STATE.OP, E_LAMP_SUBSTATE.OP_WARMING);
			RETURN;
		ELSIF nEvent = E_LAMP_EVENT.WARMED_UP THEN
			// This event will happen if there is no warmup. 
			// We go directly to ON.
			SetState(E_LAMP_STATE.OP, E_LAMP_SUBSTATE.OP_ON);
			RETURN;				
		ELSIF nEvent = E_LAMP_EVENT.ON THEN
			// Another Lamp ON command received while switching ON
			M_UpdateCtrlParams();
			// Restart the TimeON
			M_UpdateTimes(bOnState:=TRUE,bRestart:=TRUE, bReset:=FALSE);
			RETURN;
		ELSIF nEvent = E_LAMP_EVENT.ERRTIMEOUTON  THEN
			// Timeout means that the lamp is still off.
			// The error has been set in ActivitySwitchingOn().
			SetState(E_LAMP_STATE.OP, E_LAMP_SUBSTATE.OP_OFF);
			RETURN;
		END_IF
		
	E_LAMP_SUBSTATE.OP_WARMING:			
		IF nEvent = E_LAMP_EVENT.OFF  OR  nEvent = E_LAMP_EVENT.LIMIT_ON THEN
			ActionOffExecute();
			SetState(E_LAMP_STATE.OP, E_LAMP_SUBSTATE.OP_SWITCHING_OFF);
			RETURN;
		ELSIF nEvent = E_LAMP_EVENT.ON THEN
			// Another Lamp ON command received while warming up
			M_UpdateCtrlParams();
			// Restart the TimeON
			M_UpdateTimes(bOnState:=TRUE,bRestart:=TRUE, bReset:=FALSE);
			RETURN;
		ELSIF nEvent = E_LAMP_EVENT.ISOFF THEN
			ActionUnexpExecute();
			SetState(E_LAMP_STATE.OP, E_LAMP_SUBSTATE.OP_OFF);
			RETURN;
		ELSIF nEvent = E_LAMP_EVENT.DISABLE THEN
			ActionDisableExecute();
			SetState(E_LAMP_STATE.OP, E_LAMP_SUBSTATE.OP_DISABLING);
			RETURN;	
		ELSIF nEvent = E_LAMP_EVENT.STOP THEN
			ActionOffExecute();
			SetState(E_LAMP_STATE.OP, E_LAMP_SUBSTATE.OP_SWITCHING_OFF);
			RETURN;
		ELSIF nEvent = E_LAMP_EVENT.WARMED_UP THEN
			SetState(E_LAMP_STATE.OP, E_LAMP_SUBSTATE.OP_ON);
			RETURN;				
		ELSIF nEvent = E_LAMP_EVENT.ERRMAXON THEN
			ActionMaxOnFailure();
			SetState(E_LAMP_STATE.OP, E_LAMP_SUBSTATE.OP_SWITCHING_OFF);
			RETURN;				
		END_IF
		
	E_LAMP_SUBSTATE.OP_ON:			
		IF nEvent = E_LAMP_EVENT.OFF  OR  nEvent = E_LAMP_EVENT.LIMIT_ON	THEN
			ActionOffExecute();
			SetState(E_LAMP_STATE.OP, E_LAMP_SUBSTATE.OP_SWITCHING_OFF);
			RETURN;
		ELSIF nEvent = E_LAMP_EVENT.ON THEN
			M_LogEventGeneral('New ON command while ON.');
			// Clear previous error, if any.
			M_SetStatus(E_LAMP_ERROR.OK);
			M_UpdateCtrlParams();
			// Restart the TimeON
			M_UpdateTimes(bOnState:=TRUE,bRestart:=TRUE, bReset:=FALSE);
			RETURN;
		ELSIF nEvent = E_LAMP_EVENT.ISOFF THEN
			ActionUnexpExecute();
			SetState(E_LAMP_STATE.OP, E_LAMP_SUBSTATE.OP_OFF);
			RETURN;
		ELSIF nEvent = E_LAMP_EVENT.DISABLE THEN
			ActionDisableExecute();
			SetState(E_LAMP_STATE.OP, E_LAMP_SUBSTATE.OP_DISABLING);
			RETURN;	
		ELSIF nEvent = E_LAMP_EVENT.ERRMAXON THEN
			ActionMaxOnFailure();
			SetState(E_LAMP_STATE.OP, E_LAMP_SUBSTATE.OP_SWITCHING_OFF);
			RETURN;				
		END_IF
		
	E_LAMP_SUBSTATE.OP_SWITCHING_OFF:			
		IF nEvent = E_LAMP_EVENT.ISOFF THEN
			// This event will happen if there is cooldown
			SetState(E_LAMP_STATE.OP, E_LAMP_SUBSTATE.OP_COOLING);
			RETURN;
		ELSIF nEvent = E_LAMP_EVENT.COOLED_DOWN THEN
			// This event will happen if there is no cooldown. 
			// We go directly to OFF.
			SetState(E_LAMP_STATE.OP, E_LAMP_SUBSTATE.OP_OFF);
			RETURN;				
		ELSIF nEvent = E_LAMP_EVENT.ERRTIMEOUTOFF  THEN
			SetState(E_LAMP_STATE.OP, E_LAMP_SUBSTATE.OP_OFF);
			RETURN;
		END_IF
		
	E_LAMP_SUBSTATE.OP_COOLING:			
		IF nEvent = E_LAMP_EVENT.ON THEN
			ActionUnexpExecute();
			//SetState(E_LAMP_STATE.OP, E_LAMP_SUBSTATE.OP_ERROR);
			RETURN;
		ELSIF nEvent = E_LAMP_EVENT.ISON THEN
			ActionUnexpExecute();
			SetState(E_LAMP_STATE.OP, E_LAMP_SUBSTATE.OP_ON);
			RETURN;
		ELSIF nEvent = E_LAMP_EVENT.DISABLE THEN
			ActionDisableExecute();
			SetState(E_LAMP_STATE.OP, E_LAMP_SUBSTATE.OP_DISABLING);
			RETURN;	
		ELSIF nEvent = E_LAMP_EVENT.COOLED_DOWN THEN
			SetState(E_LAMP_STATE.OP, E_LAMP_SUBSTATE.OP_OFF);
			RETURN;				
		END_IF
		
	E_LAMP_SUBSTATE.OP_ERROR:			
		IF nEvent = E_LAMP_EVENT.OFF THEN
			ActionOffExecute();
			SetState(E_LAMP_STATE.OP, E_LAMP_SUBSTATE.OP_SWITCHING_OFF);
			RETURN;
		ELSIF nEvent = E_LAMP_EVENT.ON THEN
			ActionOnExecute();
			SetState(E_LAMP_STATE.OP, E_LAMP_SUBSTATE.OP_SWITCHING_ON);
			RETURN;			
		ELSIF nEvent = E_LAMP_EVENT.ISON THEN
			M_LogEventGeneral('Recovered from error. Lamp is ON.');
			SetState(E_LAMP_STATE.OP, E_LAMP_SUBSTATE.OP_ON);
			RETURN;			
		ELSIF nEvent = E_LAMP_EVENT.ISOFF THEN
			M_LogEventGeneral('Recovered from error. Lamp is OFF.');
			SetState(E_LAMP_STATE.OP, E_LAMP_SUBSTATE.OP_OFF);
			RETURN;	
		ELSIF nEvent = E_LAMP_EVENT.DISABLE THEN
			SetState(E_LAMP_STATE.OP, E_LAMP_SUBSTATE.OP_DISABLING);
			RETURN;			
		END_IF

	E_LAMP_SUBSTATE.OP_DISABLING:			
		IF nEvent = E_LAMP_EVENT.DISABLEOFF THEN
			M_UpdateTimes(bOnState:=FALSE,bRestart:=FALSE, bReset:=FALSE);	// Update the Time
			SetState(E_LAMP_STATE.NOTOP, E_LAMP_SUBSTATE.NOTOP_READY_OFF);
			RETURN;
		ELSIF nEvent = E_LAMP_EVENT.DISABLEON THEN
			M_UpdateTimes(bOnState:=TRUE,bRestart:=FALSE, bReset:=FALSE);	// Update the Time
			SetState(E_LAMP_STATE.NOTOP, E_LAMP_SUBSTATE.NOTOP_READY_ON);
			RETURN;
		ELSIF nEvent = E_LAMP_EVENT.ERRDISABLE THEN
			SetState(E_LAMP_STATE.NOTOP, E_LAMP_SUBSTATE.NOTOP_NOTREADY);
			RETURN;
		END_IF
		
	END_CASE
	
	(* Transitions from any OP substate *)
	IF nEvent = E_LAMP_EVENT.ERRHW THEN
		SetState(E_LAMP_STATE.OP, E_LAMP_SUBSTATE.OP_ERROR);
		RETURN;
	ELSIF nEvent = E_LAMP_EVENT.ERRFAULT THEN
		ActionErrExecute();
		SetState(E_LAMP_STATE.OP, E_LAMP_SUBSTATE.OP_ERROR);
		RETURN;				
	ELSIF nEvent = E_LAMP_EVENT.RESET THEN
		ActionResetExecute();
		SetState(E_LAMP_STATE.NOTOP, E_LAMP_SUBSTATE.NOTOP_NOTREADY);
		RETURN;
	END_IF
	
END_CASE

(* 
	"Global" internal transitions valid in any state should go here.
	They do not change the active state configuration. 
	They are evaluated after all the others transitions have been 
	considered.
*) 
IF nEvent = E_LAMP_EVENT.STOP THEN
	RETURN;
END_IF
END_METHOD

METHOD SetAction
VAR_INPUT
	actionName:		STRING;
END_VAR


stat.sActionDesc := actionName;
END_METHOD

METHOD SetEvent
VAR_INPUT
	nEventId:			DINT;
END_VAR
// Set the event
nEvent := nEventId;

// Set the textual description of the event
CASE nEventId OF
	E_LAMP_EVENT.NONE:
		stat.sEventDesc := '';
		RETURN;
		
	E_LAMP_EVENT.RESET:
		stat.sEventDesc := 'CMD RESET';
		RETURN;
	
	E_LAMP_EVENT.INIT:
		stat.sEventDesc := 'CMD INIT';
		RETURN;

	E_LAMP_EVENT.STOP:
		stat.sEventDesc := 'CMD STOP';
		RETURN;

	E_LAMP_EVENT.ENABLE:
		stat.sEventDesc := 'CMD ENABLE';
		RETURN;

	E_LAMP_EVENT.DISABLE:
		stat.sEventDesc := 'CMD DISABLE';
		RETURN;

	E_LAMP_EVENT.ON:
		stat.sEventDesc := 'CMD ON';
		RETURN;

	E_LAMP_EVENT.OFF:
		stat.sEventDesc := 'CMD OFF';
		RETURN;
	
	(* events corresponding to internal events *)
	E_LAMP_EVENT.INITOFF:
		stat.sEventDesc := 'INT INITOFF';
		RETURN;

	E_LAMP_EVENT.INITON:
		stat.sEventDesc := 'INT INITON';
		RETURN;

	E_LAMP_EVENT.DISABLEOFF:
		stat.sEventDesc := 'INT DISABLEOFF';
		RETURN;
	
	E_LAMP_EVENT.DISABLEON:
		stat.sEventDesc := 'INT DISABLEON';
		RETURN;
	
	(* evetnts mapped to HW signals *)
	E_LAMP_EVENT.ISON:
		stat.sEventDesc := 'SIG ISON';
		RETURN;

	E_LAMP_EVENT.WARMED_UP:
		stat.sEventDesc := 'INT WARMED UP';
		RETURN;

	E_LAMP_EVENT.COOLED_DOWN:
		stat.sEventDesc := 'INT COOLED DOWN';
		RETURN;

	E_LAMP_EVENT.LIMIT_ON:
		stat.sEventDesc := 'INT TIME ON LIMIT';
		RETURN;

	E_LAMP_EVENT.ISOFF:
		stat.sEventDesc := 'SIG ISOFF';
		RETURN;

	E_LAMP_EVENT.HWOK:
		stat.sEventDesc := 'SIG HWOK';
		RETURN;

	E_LAMP_EVENT.ERRHW:
		stat.sEventDesc := 'INT ERRHW';
		RETURN;

	E_LAMP_EVENT.ERRMAXON:
		stat.sEventDesc := 'INT ERRMAXON';
		RETURN;

	E_LAMP_EVENT.ERRFAULT:	
		stat.sEventDesc := 'INT ERRFAULT';
		RETURN;

	E_LAMP_EVENT.ERRINIT:
		stat.sEventDesc := 'INT ERRINIT';
		RETURN;

	E_LAMP_EVENT.ERRDISABLE:
		stat.sEventDesc := 'INT ERRDISABLE';
		RETURN;
	
	E_LAMP_EVENT.ERRTIMEOUTOFF:
		stat.sEventDesc := 'INT ERRTIMEOUTOFF';
		RETURN;
	
	E_LAMP_EVENT.ERRTIMEOUTON:
		stat.sEventDesc := 'INT ERRTIMEOUTON';
		RETURN;
	
END_CASE 

(* INTERNAL ERROR *)
stat.sEventDesc := 'UNKNOWN EVENT';
END_METHOD

METHOD SetState : BOOL
VAR_INPUT
	nState:			E_LAMP_STATE;
	nSubstate:		E_LAMP_SUBSTATE;
END_VAR
(* 
	Update State Machine active state configuration.

	ToDo: support initial pseudo state/substate.
*)

IF nState <> E_LAMP_STATE.NONE THEN
	stat.nState	:= nState;
END_IF
IF nSubstate <> E_LAMP_SUBSTATE.NONE THEN
	stat.nSubstate	:= nSubstate;
END_IF

(* Update active state configuration description *)

IF nState = E_LAMP_STATE.NOTOP THEN
	stat.sState	:= 'NOT OP';
ELSIF nState = E_LAMP_STATE.OP THEN
	stat.sState	:= 'OPERATIONAL';
END_IF

IF nSubstate = E_LAMP_SUBSTATE.NOTOP_NOTREADY THEN
	stat.sSubstate	:= 'NOT READY';
ELSIF nSubstate = E_LAMP_SUBSTATE.NOTOP_INITIALIZING THEN
	stat.sSubstate	:= 'INITIALIAZING';
ELSIF nSubstate = E_LAMP_SUBSTATE.NOTOP_READY_OFF THEN
	stat.sSubstate	:= 'READY OFF';
ELSIF nSubstate = E_LAMP_SUBSTATE.NOTOP_READY_ON THEN
	stat.sSubstate	:= 'READY ON';
ELSIF nSubstate = E_LAMP_SUBSTATE.NOTOP_ERROR THEN
	stat.sSubstate	:= 'ERROR';
ELSIF nSubstate = E_LAMP_SUBSTATE.OP_OFF THEN
	stat.sSubstate	:= 'OFF';
ELSIF nSubstate = E_LAMP_SUBSTATE.OP_ON THEN
	stat.sSubstate	:= 'ON';
ELSIF nSubstate = E_LAMP_SUBSTATE.OP_SWITCHING_OFF THEN
	stat.sSubstate	:= 'SWITCHING OFF';
ELSIF nSubstate = E_LAMP_SUBSTATE.OP_SWITCHING_ON THEN
	stat.sSubstate	:= 'SWITCHING ON';
ELSIF nSubstate = E_LAMP_SUBSTATE.OP_WARMING THEN
	stat.sSubstate	:= 'WARMING UP';
ELSIF nSubstate = E_LAMP_SUBSTATE.OP_COOLING THEN
	stat.sSubstate	:= 'COOLING DOWN';
ELSIF nSubstate = E_LAMP_SUBSTATE.OP_DISABLING THEN
	stat.sSubstate	:= 'DISABLING';
ELSIF nSubstate = E_LAMP_SUBSTATE.OP_ERROR THEN
	stat.sSubstate	:= 'ERROR';
ELSE
	stat.sSubstate	:= '';
END_IF


SetState	:= TRUE;
END_METHOD

END_FUNCTION_BLOCK

// ---- POUs/MAIN.TcPOU
PROGRAM MAIN
VAR
	// Lamp instances
	{attribute 'OPC.UA.DA':='1'}
	Lamp001:		FB_LAMP;	
	{attribute 'OPC.UA.DA':='1'}
	Lamp002:		FB_LAMP;	
	
	// Simulators
	{attribute 'OPC.UA.DA':='1'}
	SIM_Lamp001:	FB_SIM_LAMP;
	{attribute 'OPC.UA.DA':='1'}
	SIM_Lamp002:	FB_SIM_LAMP;
END_VAR

Lamp001(in_sName:='Lamp001', in_nTimeout:=5000);
Lamp002(in_sName:='Lamp002', in_nTimeout:=3000, in_nCooldown:=5, in_nMaxOn:=30);

SIM_Lamp001(ptrDev:=ADR(Lamp001));
SIM_Lamp002(ptrDev:=ADR(Lamp002));

END_PROGRAM

// ---- GlobalTextList.TcGTLO
TEXTLIST GlobalTextList
  46 = '%.0f'
  23 = '%d'
  62 = '%d sec '
  13 = '%s'
  464 = "'IODev.library version'"
  77 = 'A period of time [ms] that the feedback signal has to have constant value before taking its status.'
  78 = 'A period of time [ms] that the feedback signal has to have constant value before taking its status.\nMinimum 10 ms.'
  246 = 'Absolut maximum allowed time for lamp to be ON after last ON command [sec]  (>=0). \nZero means no limit.\n'
  766 = 'Absolut maximum allowed time for lamp to be ON after last ON command [sec]  (>=0). \nZero means no limit.\nThis is a safety feature.\n'
  26 = 'Action'
  8 = 'ACTIVATE'
  36 = 'Active Low'
  67 = 'Actual Lamp intensity [%] (0..100)'
  357 = 'Actual Time ON limit [sec]'
  70 = 'Analog feedback signal threshold [bit].\nIf used, the threshold should be > 0.\n'
  263 = 'Analog feedback [bit]'
  92 = 'Analog Feedback [bit]'
  71 = 'AnalogThreshold [bit]'
  516 = 'Anlg Fdbk [bit]'
  1005 = 'Anlg Feedback [bit]'
  91 = 'Auto OFF after this time [sec]. 0 - no limit'
  39 = 'Checkbox'
  15 = 'CLOSE'
  35 = 'Configuration'
  56 = 'Control'
  58 = 'Cooldown'
  53 = 'Cooldown time [sec]  (>=0). \nZero means no cooldown.\n'
  50 = 'Cooldown [sec]'
  9 = 'DEACTIVATE'
  108 = 'Device Status\n0 - OK\n1 - FAILURE'
  7 = 'DISABLE'
  6 = 'ENABLE'
  74 = 'Error Code'
  190 = 'Error Code\n0 - OK'
  19 = 'Error Description'
  27 = 'Event'
  40 = 'Fault'
  297 = 'Feedback Timeout [ms]'
  73 = 'Feedback Timeout [sec]'
  63 = 'Full range of A/D converter controlling the intensity [bit]  (>=0). \n'
  55 = 'Full range of A/D converter controlling the intensity [bit].\nExamples:\n12 bit A/D = 4095\n15 bit A/D = 32767 \n16 bit A/D = 65535\n'
  52 = 'Full range [bit]'
  61 = 'GREEN means state is active'
  69 = 'GUI disabled !!!\nActivate "Local Control".'
  22 = 'HW'
  28 = 'HW Status'
  269 = 'If ON, check for maximum time is active.'
  931 = 'If ON, digital control output is active'
  89 = 'If ON, digital control output is high.'
  557 = 'If ON, digital control output isignal s high (TRUE)'
  567 = 'If ON, Fault signal is active.'
  146 = 'If ON, Fault signal is high (TRUE).'
  540 = 'If ON, Fault signal is high.'
  833 = 'If ON, Lamp Analog feedback signal is active.'
  792 = 'If ON, Lamp Digital feedback signal is high (TRUE).'
  860 = 'If ON, Lamp ON feedback signal is active.'
  319 = 'If ON, Lamp ON signal is active.'
  705 = 'If ON, Open switch is active.'
  1111 = 'If selected, the lamp will switch ON on INIT.'
  44 = 'If the logic is inverted, the lamp is considered to be ON, if the reading is below the threshold.'
  37 = 'Ignore'
  38 = 'Ignore Fault'
  4 = 'INIT'
  951 = 'Initial Intensity [%]'
  162 = 'Initial State'
  64 = 'Intensity [%]'
  43 = 'Inver Analog Logic'
  45 = 'Invert Analog Logic'
  132 = 'Invert Logic'
  16 = 'ISOPEN'
  66 = 'Lamp has to be initialised before it can be used.\n\nRED = not initialised\nGREEN = initialised\n'
  355 = 'Lamp will stay ON for this time [sec] and will automatically switch OFF. \nZero means no limit.'
  65 = 'Local Control'
  411 = 'Log'
  51 = 'Max ON [sec]'
  54 = 'Maximum allowed time for lamp to be ON [sec]  (>=0). \nZero means no limit.\n'
  17 = 'not used'
  30 = 'OFF'
  29 = 'ON'
  41 = 'On'
  90 = 'ON Limit [sec]'
  14 = 'OPEN'
  60 = 'ORANGE means state is active'
  10 = 'POWER OFF'
  59 = 'RED means state is active'
  192 = 'Remaining  [sec]'
  1082 = 'Remaining time before the Lamp is switched OFF [sec].'
  3 = 'RESET'
  2 = 'REST'
  941 = 'RPC Call Status'
  578 = 'RPC Error Code'
  561 = 'RPC Error Code\n0 - OK'
  47 = 'Set Lamp intensity [%] (0..100)'
  956 = 'Set limit for Lamp to stay ON [sec] and automatically switch OFF. \nZero means no limit.'
  740 = 'Set value for limit for Lamp to stay ON [sec] and automatically switch OFF. \nZero means no limit.'
  75 = 'Stable Signal Period'
  76 = 'Stable Signal Period [ms]'
  11 = 'STATE'
  24 = 'State'
  0 = 'State: %s'
  18 = 'STATUS'
  20 = 'Status'
  21 = 'Status Description'
  5 = 'STOP'
  12 = 'SUBSTATE'
  25 = 'Substate'
  1 = 'Substate: %s'
  42 = 'Switch'
  381 = 'Switch logging ON/OFF'
  33 = 'Time OFF = %d'
  34 = 'Time OFF Total = %d'
  83 = 'Time ON'
  86 = 'Time ON  [sec]'
  31 = 'Time ON = %d'
  32 = 'Time ON Total = %d'
  82 = 'Time since Lamp was switched OFF [sec].'
  81 = 'Time since last ON command [sec].'
  79 = 'Time since last ON command.'
  80 = 'Total continuous time that Lamp has been ON [sec].'
  85 = 'Total OFF'
  88 = 'Total OFF [sec]'
  84 = 'Total ON'
  87 = 'Total ON  [sec]'
  68 = 'Ver. %.2f'
  463 = 'Ver: %s'
  57 = 'Warmup'
  48 = 'Warmup time [sec]  (>=0). \nZero means no warmup.\n'
  49 = 'Warmup [sec]'
  72 = 'When switching lamp ON, feedback signal should become active within this period.\n'
END_TEXTLIST

// ---- VISUs/GUI_Lamp001.TcVIS
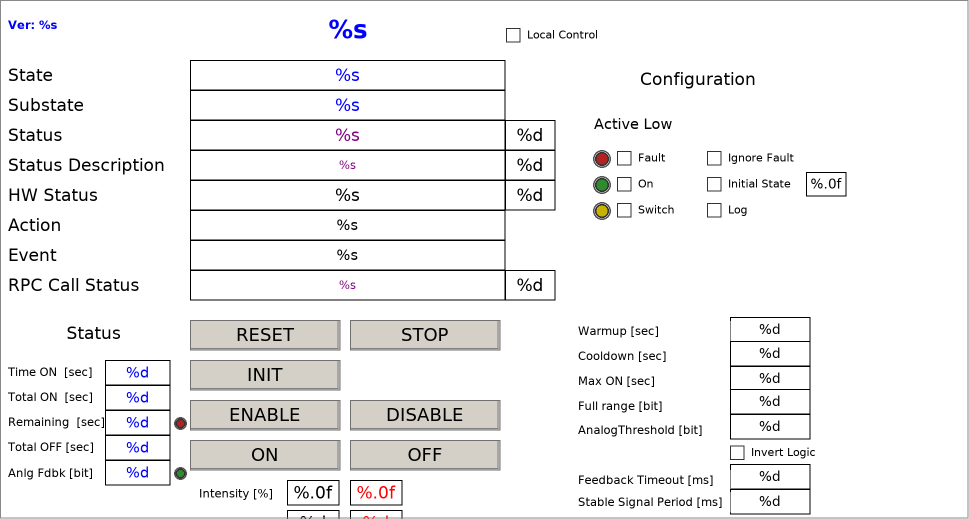
VISUALIZATION GUI_Lamp001  // 969x519
    Frame (0,0 967x517)
        shows GUI_TEMPLATE_LAMP(m_Instance := MAIN.Lamp001)
END_VISUALIZATION

// ---- VISUs/GUI_Lamp002.TcVIS
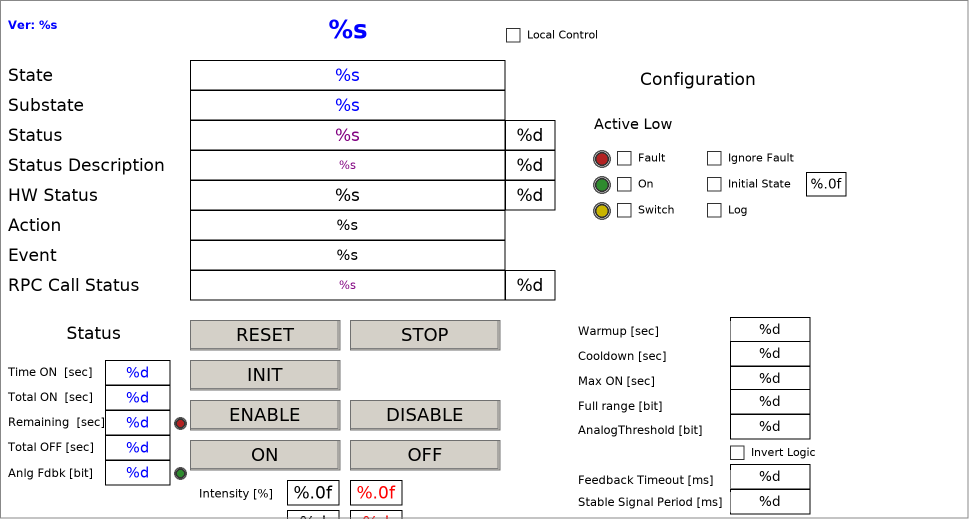
VISUALIZATION GUI_Lamp002  // 969x519
    Frame (0,0 967x517)
        shows GUI_TEMPLATE_LAMP(m_Instance := MAIN.Lamp002)
END_VISUALIZATION

// ---- VISUs/Templates/GUI_TEMPLATE_LAMP.TcVIS
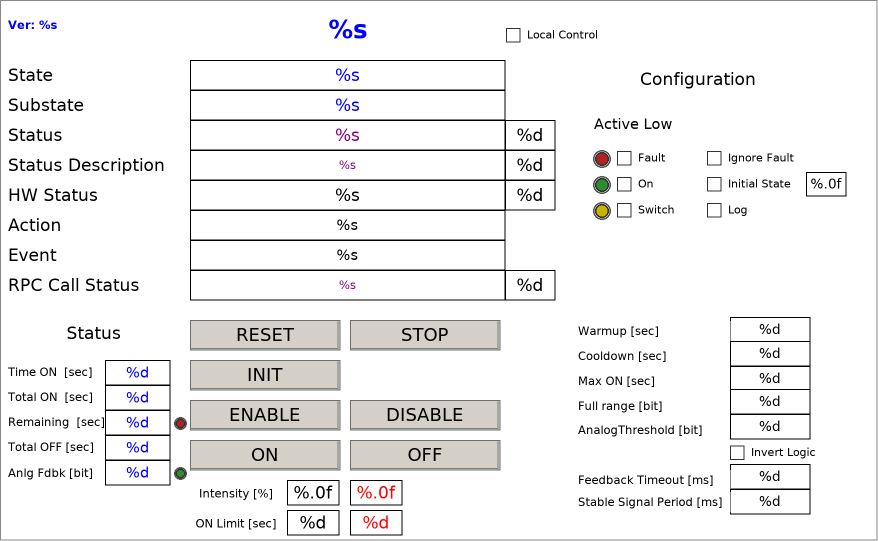
VISUALIZATION GUI_TEMPLATE_LAMP  // 878x541
VAR_IN_OUT
	m_Instance:	FB_LAMP;
END_VAR
    Rectangle (190,60 315x30), "%s", text variable: m_Instance.stat.sState
    Rectangle (190,90 315x30), "%s", text variable: m_Instance.stat.sSubstate
    Button (190,320 150x30), "RESET", input disabled if: (m_Instance.stat.bLocal = FALSE) <> 0
        OnMouseDown: execute { m_Instance.ctrl.nCommand := E_LAMP_COMMAND.RESET; m_Instance.ctrl.bExecute := TRUE; }
    Button (190,360 150x30), "INIT", input disabled if: (m_Instance.stat.bLocal = FALSE) <> 0
        OnMouseDown: execute { m_Instance.ctrl.nCommand := E_LAMP_COMMAND.INIT; m_Instance.ctrl.bExecute := TRUE; }
    Button (350,320 150x30), "STOP", input disabled if: (m_Instance.stat.bLocal = FALSE) <> 0
        OnMouseDown: execute { m_Instance.ctrl.nCommand := E_LAMP_COMMAND.STOP; m_Instance.ctrl.bExecute := TRUE; }
    Button (190,400 150x30), "ENABLE", input disabled if: (m_Instance.stat.bLocal = FALSE) <> 0
        OnMouseDown: execute { m_Instance.ctrl.nCommand := E_LAMP_COMMAND.ENABLE; m_Instance.ctrl.bExecute := TRUE; }
    Button (350,400 150x30), "DISABLE", input disabled if: (m_Instance.stat.bLocal = FALSE) <> 0
        OnMouseDown: execute { m_Instance.ctrl.nCommand := E_LAMP_COMMAND.DISABLE; m_Instance.ctrl.bExecute := TRUE; }
    Button (190,440 150x30), "ON", input disabled if: (m_Instance.stat.bLocal = FALSE) <> 0
        OnMouseDown: execute { m_Instance.ctrl.nCommand := E_LAMP_COMMAND.ON; m_Instance.ctrl.bExecute := TRUE; }
    Button (350,440 150x30), "OFF", input disabled if: (m_Instance.stat.bLocal = FALSE) <> 0
        OnMouseDown: execute { m_Instance.ctrl.nCommand := E_LAMP_COMMAND.OFF; m_Instance.ctrl.bExecute := TRUE; }
    Rectangle (5,60 180x30), "State"
    Rectangle (5,90 180x30), "Substate"
    Rectangle (190,120 315x30), "%s", text variable: m_Instance.stat.sStatus
    Rectangle (190,150 315x30), "%s", text variable: m_Instance.stat.sErrorText
    Rectangle (5,120 180x30), "Status"
    Rectangle (5,150 180x30), "Status Description"
    Rectangle (190,210 315x30), "%s", text variable: m_Instance.stat.sActionDesc
    Rectangle (190,240 315x30), "%s", text variable: m_Instance.stat.sEventDesc
    Rectangle (190,180 315x30), "%s", text variable: m_Instance.stat.sHwStatus
    Rectangle (5,180 180x30), "HW Status"
    Rectangle (505,180 50x30), "%d", text variable: m_Instance.stat.nHwStatus
    Rectangle (5,210 180x30), "Action"
    Rectangle (5,240 180x30), "Event"
    Rectangle (232,12 232x35), "%s", text variable: m_Instance.cfg.sName
    Rectangle (637,64 180x30), "Configuration"
    Rectangle (591,109 126x30), "Active Low"
    Checkbox (615,143 72x30), "Fault", variable: m_Instance.cfg.bActiveLowFault, input disabled if: (m_Instance.stat.bLocal = FALSE) <> 0
    Checkbox (705,143 102x30), "Ignore Fault", variable: m_Instance.cfg.bIgnoreFault, input disabled if: (m_Instance.stat.bLocal = FALSE) <> 0
    Checkbox (615,169 72x30), "On", variable: m_Instance.cfg.bActiveLowOn, input disabled if: (m_Instance.stat.bLocal = FALSE) <> 0
    Checkbox (615,195 72x30), "Switch", variable: m_Instance.cfg.bActiveLowSwitch, input disabled if: (m_Instance.stat.bLocal = FALSE) <> 0
    Checkbox (728,440 150x25), "Invert Logic", tooltip "If the logic is inverted, the lamp is considered to be ON, if the reading is below the threshold.", variable: m_Instance.cfg.bInvertAnalog, input disabled if: (m_Instance.stat.bLocal = FALSE) <> 0
    Rectangle (730,317 80x25), "%d", tooltip "Warmup time [sec] (>=0). Zero means no warmup.", text variable: m_Instance.cfg.nWarmup, input disabled if: (m_Instance.stat.bLocal = FALSE) <> 0
        OnMouseDown: write the text variable via Default, min 0
    Rectangle (575,321 155x20), "Warmup [sec]"
    Rectangle (575,346 155x20), "Cooldown [sec]"
    Rectangle (575,371 155x20), "Max ON [sec]"
    Rectangle (575,396 155x20), "Full range [bit]"
    Rectangle (730,341 80x25), "%d", tooltip "Cooldown time [sec] (>=0). Zero means no cooldown.", text variable: m_Instance.cfg.nCooldown, input disabled if: (m_Instance.stat.bLocal = FALSE) <> 0
        OnMouseDown: write the text variable via Default, min 0
    Rectangle (730,366 80x25), "%d", tooltip "Absolut maximum allowed time for lamp to be ON after last ON command [sec] (>=0). Zero means no limit. This is a safety feature.", text variable: m_Instance.cfg.nMaxOn, input disabled if: (m_Instance.stat.bLocal = FALSE) <> 0
        OnMouseDown: write the text variable via Default, min 0
    Rectangle (730,389 80x25), "%d", tooltip "Full range of A/D converter controlling the intensity [bit]. Examples: 12 bit A/D = 4095 15 bit A/D = 32767 16 bit A/D = 65535", text variable: m_Instance.cfg.nFullRange, input disabled if: (m_Instance.stat.bLocal = FALSE) <> 0
        OnMouseDown: write the text variable via Default, min 0
    Rectangle (730,414 80x25), "%d", tooltip "Analog feedback signal threshold [bit]. If used, the threshold should be > 0.", text variable: m_Instance.cfg.nAnalogThreshold, input disabled if: (m_Instance.stat.bLocal = FALSE) <> 0
        OnMouseDown: write the text variable via Default, min 0
    Rectangle (575,420 150x20), "AnalogThreshold [bit]"
    Rectangle (730,464 80x25), "%d", tooltip "When switching lamp ON, feedback signal should become active within this period.", text variable: m_Instance.cfg.nTimeout, input disabled if: (m_Instance.stat.bLocal = FALSE) <> 0
        OnMouseDown: write the text variable via Default, min 0
    Rectangle (575,470 155x20), "Feedback Timeout [ms]"
    Rectangle (287,480 52x25), "%.0f", tooltip "Set Lamp intensity [%] (0..100)", text variable: m_Instance.ctrl.lrIntensity, input disabled if: (m_Instance.stat.bLocal = FALSE) <> 0
        OnMouseDown: write the text variable via Default, min 0
    Rectangle (191,476 90x35), "Intensity [%]"
    Rectangle (350,480 52x25), "%.0f", tooltip "Actual Lamp intensity [%] (0..100)", text variable: m_Instance.stat.lrIntensity
    Checkbox (504,20 116x30), "Local Control", variable: m_Instance.stat.bLocal
    Rectangle (730,489 80x25), "%d", tooltip "A period of time [ms] that the feedback signal has to have constant value before taking its status. Minimum 10 ms.", text variable: m_Instance.cfg.nSigStablePeriod, input disabled if: (m_Instance.stat.bLocal = FALSE) <> 0
        OnMouseDown: write the text variable via Default, min 10
    Rectangle (575,492 155x20), "Stable Signal Period [ms]"
    Rectangle (48,318 92x30), "Status"
    Rectangle (105,360 65x25), "%d", tooltip "Time since last ON command [sec].", text variable: m_Instance.stat.nTimeOn
    Rectangle (105,385 65x25), "%d", tooltip "Total continuous time that Lamp has been ON [sec].", text variable: m_Instance.stat.nTimeOnTotal
    Rectangle (105,435 65x25), "%d", tooltip "Time since Lamp was switched OFF [sec].", text variable: m_Instance.stat.nTimeOff
    Rectangle (5,357 95x30), "Time ON [sec]"
    Rectangle (5,382 95x30), "Total ON [sec]"
    Rectangle (5,432 95x30), "Total OFF [sec]"
    Rectangle (505,120 50x30), "%d", tooltip "Device Status 0 - OK 1 - FAILURE", text variable: m_Instance.stat.nStatus
    Rectangle (190,270 315x30), "%s", text variable: m_Instance.stat.sRpcErrorText
    Rectangle (5,270 180x30), "RPC Call Status"
    Rectangle (5,10 99x30), "Ver: %s", tooltip "'IODev.library version'", text variable: m_Instance.stat.sLibVersion, input disabled if: true
    Rectangle (505,270 50x30), "%d", tooltip "RPC Error Code 0 - OK", text variable: m_Instance.stat.nRpcErrorCode
    Rectangle (505,150 50x30), "%d", tooltip "Error Code 0 - OK", text variable: m_Instance.stat.nErrorCode
    Lamp1 (592,149 20x20), tooltip "If ON, Fault signal is high (TRUE).", variable: m_Instance.i_bFault, style: Lamp-Lamp1-Red
    Lamp1 (592,201 20x20), tooltip "If ON, digital control output isignal s high (TRUE)", variable: m_Instance.q_bSwitch, style: Lamp-Lamp1-Yellow
    Lamp1 (592,175 20x20), tooltip "If ON, Lamp Digital feedback signal is high (TRUE).", variable: m_Instance.i_bOn, style: Lamp-Lamp1-Green
    Rectangle (287,510 52x25), "%d", tooltip "Set value for limit for Lamp to stay ON [sec] and automatically switch OFF. Zero means no limit.", text variable: m_Instance.ctrl.nTimeOnLimit, input disabled if: (m_Instance.stat.bLocal = FALSE) <> 0
        OnMouseDown: write the text variable via Default, min 0
    Rectangle (191,506 90x35), "ON Limit [sec]"
    Rectangle (350,510 52x25), "%d", tooltip "Actual Time ON limit [sec]", text variable: m_Instance.stat.nTimeOnLimit
    Rectangle (5,407 97x30), "Remaining [sec]"
    Rectangle (105,410 65x25), "%d", tooltip "Remaining time before the Lamp is switched OFF [sec].", text variable: m_Instance.stat.nTimeLeft
    Lamp1 (173,416 15x15), tooltip "If ON, check for maximum time is active.", variable: m_Instance.stat.bCheckTimeLeft, style: Lamp-Lamp1-Red
    Checkbox (705,169 100x30), "Initial State", tooltip "If selected, the lamp will switch ON on INIT.", variable: m_Instance.cfg.bInitialState, input disabled if: (m_Instance.stat.bLocal = FALSE) <> 0
    Rectangle (806,172 40x24), "%.0f", tooltip "Initial Intensity [%]", text variable: m_Instance.cfg.lrInitialIntensity, input disabled if: (m_Instance.stat.bLocal = FALSE) <> 0
        OnMouseDown: write the text variable via Default, min 0
    Checkbox (705,195 95x30), "Log", tooltip "Switch logging ON/OFF", variable: m_Instance.cfg.bLog, input disabled if: (m_Instance.stat.bLocal = FALSE) <> 0
    Lamp1 (173,466 15x15), tooltip "If ON, Lamp Analog feedback signal is active.", variable: m_Instance.stat.bOnAnalog, style: Lamp-Lamp1-Green
    Rectangle (105,460 65x25), "%d", tooltip "Analog Feedback [bit]", text variable: m_Instance.stat.nOn
    Rectangle (5,458 95x30), "Anlg Fdbk [bit]", tooltip "Analog Feedback [bit]"
END_VISUALIZATION
